LIN {X 0,Y 573.254,Z 377.707,A -85,B 0,C 180,E1 -2096.976,E2 -2096.976} C_VEL
LIN {X 0,Y 573.253,Z 377.7,A -85,B 0,C 180,E1 -2099.488,E2 -2099.488} C_VEL
LIN {X 0,Y 573.258,Z 377.706,A -85,B 0,C 180,E1 -2102.645,E2 -2102.645} C_VEL
LIN {X 0,Y 573.214,Z 377.706,A -85,B 0,C 180,E1 -2105.188,E2 -2105.188} C_VEL
LIN {X 0,Y 573.24,Z 377.699,A -85,B 0,C 180,E1 -2107.808,E2 -2107.808} C_VEL
LIN {X 0,Y 573.25,Z 377.708,A -85,B 0,C 180,E1 -2110.525,E2 -2110.525} C_VEL
LIN {X 0,Y 573.244,Z 377.699,A -85,B 0,C 180,E1 -2113.359,E2 -2113.359} C_VEL
LIN {X 0,Y 573.258,Z 377.706,A -85,B 0,C 180,E1 -2116.33,E2 -2116.33} C_VEL
LIN {X 0,Y 573.264,Z 377.696,A -85,B 0,C 180,E1 -2119.476,E2 -2119.476} C_VEL
LIN {X 0,Y 573.242,Z 377.706,A -85,B 0,C 180,E1 -2122.193,E2 -2122.193} C_VEL
LIN {X 0,Y 573.257,Z 377.698,A -85,B 0,C 180,E1 -2124.815,E2 -2124.815} C_VEL
LIN {X 0,Y 573.258,Z 377.698,A -85,B 0,C 180,E1 -2127.355,E2 -2127.355} C_VEL
LIN {X 0,Y 573.25,Z 377.694,A -85,B 0,C 180,E1 -2130.512,E2 -2130.512} C_VEL
LIN {X 0,Y 573.254,Z 377.697,A -85,B 0,C 180,E1 -2133.024,E2 -2133.024} C_VEL
LIN {X 0,Y 573.277,Z 377.699,A -85,B 0,C 180,E1 -2135.366,E2 -2135.366} C_VEL
LIN {X 0,Y 573.233,Z 377.701,A -85,B 0,C 180,E1 -2138.419,E2 -2138.419} C_VEL
LIN {X 0,Y 573.272,Z 377.696,A -85,B 0,C 180,E1 -2140.731,E2 -2140.731} C_VEL
LIN {X 0,Y 573.253,Z 377.706,A -85,B 0,C 180,E1 -2143.622,E2 -2143.622} C_VEL
LIN {X 0,Y 573.255,Z 377.7,A -85,B 0,C 180,E1 -2146.485,E2 -2146.485} C_VEL
LIN {X 0,Y 574.102,Z 381.406,A -85,B 0,C 180,E1 -2146.64,E2 -2146.64} C_VEL
LIN {X 0,Y 573.92,Z 396.904,A -85,B 0,C 180,E1 -2147.266,E2 -2147.266} C_VEL
LIN {X 0,Y 573.779,Z 408.749,A -85,B 0,C 180,E1 -2147.892,E2 -2147.892} C_VEL
LIN {X 0,Y 573.607,Z 419.401,A -85,B 0,C 180,E1 -2148.575,E2 -2148.575} C_VEL
LIN {X 0,Y 573.485,Z 431.28,A -85,B 0,C 180,E1 -2149.497,E2 -2149.497} C_VEL
LIN {X 0,Y 573.374,Z 441.636,A -85,B 0,C 180,E1 -2150.475,E2 -2150.475} C_VEL
LIN {X 0,Y 573.236,Z 450.947,A -85,B 0,C 180,E1 -2151.54,E2 -2151.54} C_VEL
LIN {X 0,Y 573.142,Z 458.728,A -85,B 0,C 180,E1 -2152.602,E2 -2152.602} C_VEL
LIN {X 0,Y 573.084,Z 465.205,A -85,B 0,C 180,E1 -2153.663,E2 -2153.663} C_VEL
LIN {X 0,Y 573.009,Z 470.597,A -85,B 0,C 180,E1 -2154.722,E2 -2154.722} C_VEL
LIN {X 0,Y 573.038,Z 476.255,A -85,B 0,C 180,E1 -2156.132,E2 -2156.132} C_VEL
LIN {X 0,Y 572.964,Z 479.465,A -85,B 0,C 180,E1 -2157.188,E2 -2157.188} C_VEL
LIN {X 0,Y 572.942,Z 482.451,A -85,B 0,C 180,E1 -2158.594,E2 -2158.594} C_VEL
LIN {X 0,Y 572.936,Z 484.094,A -85,B 0,C 180,E1 -2160,E2 -2160} C_VEL
LIN {X 0,Y 572.945,Z 484.433,A -85,B 0,C 180,E1 -2161.406,E2 -2161.406} C_VEL
LIN {X 0,Y 572.955,Z 483.443,A -85,B 0,C 180,E1 -2162.812,E2 -2162.812} C_VEL
LIN {X 0,Y 573.007,Z 481.089,A -85,B 0,C 180,E1 -2164.22,E2 -2164.22} C_VEL
LIN {X 0,Y 572.994,Z 478.392,A -85,B 0,C 180,E1 -2165.278,E2 -2165.278} C_VEL
LIN {X 0,Y 573.03,Z 473.984,A -85,B 0,C 180,E1 -2166.568,E2 -2166.568} C_VEL
LIN {X 0,Y 573.062,Z 468.762,A -85,B 0,C 180,E1 -2167.753,E2 -2167.753} C_VEL
LIN {X 0,Y 573.131,Z 460.802,A -85,B 0,C 180,E1 -2169.173,E2 -2169.173} C_VEL
LIN {X 0,Y 573.233,Z 451.987,A -85,B 0,C 180,E1 -2170.419,E2 -2170.419} C_VEL
LIN {X 0,Y 573.33,Z 442.788,A -85,B 0,C 180,E1 -2171.49,E2 -2171.49} C_VEL
LIN {X 0,Y 573.474,Z 431.634,A -85,B 0,C 180,E1 -2172.564,E2 -2172.564} C_VEL
LIN {X 0,Y 573.638,Z 420.168,A -85,B 0,C 180,E1 -2173.461,E2 -2173.461} C_VEL
LIN {X 0,Y 573.788,Z 409.059,A -85,B 0,C 180,E1 -2174.18,E2 -2174.18} C_VEL
LIN {X 0,Y 573.948,Z 396.515,A -85,B 0,C 180,E1 -2174.843,E2 -2174.843} C_VEL
LIN {X 0,Y 574.119,Z 381.65,A -85,B 0,C 180,E1 -2175.441,E2 -2175.441} C_VEL
LIN {X 0,Y 573.281,Z 377.703,A -85,B 0,C 180,E1 -2175.601,E2 -2175.601} C_VEL
LIN {X 0,Y 573.24,Z 377.706,A -85,B 0,C 180,E1 -2178.588,E2 -2178.588} C_VEL
LIN {X 0,Y 573.254,Z 377.705,A -85,B 0,C 180,E1 -2181.291,E2 -2181.291} C_VEL
LIN {X 0,Y 573.237,Z 377.708,A -85,B 0,C 180,E1 -2183.865,E2 -2183.865} C_VEL
LIN {X 0,Y 573.239,Z 377.709,A -85,B 0,C 180,E1 -2186.492,E2 -2186.492} C_VEL
LIN {X 0,Y 573.241,Z 377.705,A -85,B 0,C 180,E1 -2188.564,E2 -2188.564} C_VEL
LIN {X 0,Y 573.228,Z 377.707,A -85,B 0,C 180,E1 -2190.993,E2 -2190.993} C_VEL
LIN {X 0,Y 573.265,Z 377.702,A -85,B 0,C 180,E1 -2193.524,E2 -2193.524} C_VEL
LIN {X 0,Y 573.217,Z 377.709,A -85,B 0,C 180,E1 -2196.051,E2 -2196.051} C_VEL
LIN {X 0,Y 573.246,Z 377.706,A -85,B 0,C 180,E1 -2198.701,E2 -2198.701} C_VEL
LIN {X 0,Y 573.256,Z 377.707,A -85,B 0,C 180,E1 -2201.595,E2 -2201.595} C_VEL
LIN {X 0,Y 573.24,Z 377.708,A -85,B 0,C 180,E1 -2204.333,E2 -2204.333} C_VEL
LIN {X 0,Y 573.244,Z 377.707,A -85,B 0,C 180,E1 -2207.358,E2 -2207.358} C_VEL
LIN {X 0,Y 573.25,Z 377.708,A -85,B 0,C 180,E1 -2210.393,E2 -2210.393} C_VEL
LIN {X 0,Y 573.297,Z 377.786,A -85,B 0,C 180,E1 -2211.559,E2 -2211.559} C_VEL
LIN {X 0,Y 573.618,Z 382.639,A -85,B 0,C 180,E1 -2212.544,E2 -2212.544} C_VEL
LIN {X 0,Y 573.399,Z 396.627,A -85,B 0,C 180,E1 -2215.205,E2 -2215.205} C_VEL
LIN {X 0,Y 573.719,Z 413.144,A -85,B 0,C 180,E1 -2218.214,E2 -2218.214} C_VEL
LIN {X 0,Y 573.944,Z 428.097,A -85,B 0,C 180,E1 -2220.873,E2 -2220.873} C_VEL
LIN {X 0,Y 573.98,Z 435.882,A -85,B 0,C 180,E1 -2222.271,E2 -2222.271} C_VEL
LIN {X 0,Y 573.829,Z 449.3,A -85,B 0,C 180,E1 -2225.001,E2 -2225.001} C_VEL
LIN {X 0,Y 573.65,Z 462.702,A -85,B 0,C 180,E1 -2227.679,E2 -2227.679} C_VEL
LIN {X 0,Y 573.5,Z 478.001,A -85,B 0,C 180,E1 -2230.678,E2 -2230.678} C_VEL
LIN {X 0,Y 573.329,Z 493.301,A -85,B 0,C 180,E1 -2233.623,E2 -2233.623} C_VEL
LIN {X 0,Y 573.293,Z 499.756,A -85,B 0,C 180,E1 -2234.854,E2 -2234.854} C_VEL
LIN {X 0,Y 574.29,Z 505.581,A -85,B 0,C 180,E1 -2234.972,E2 -2234.972} C_VEL
LIN {X 0,Y 574.206,Z 520.02,A -85,B 0,C 180,E1 -2235.26,E2 -2235.26} C_VEL
LIN {X 0,Y 574.112,Z 533.209,A -85,B 0,C 180,E1 -2235.66,E2 -2235.66} C_VEL
LIN {X 0,Y 573.972,Z 546.119,A -85,B 0,C 180,E1 -2236.186,E2 -2236.186} C_VEL
LIN {X 0,Y 573.764,Z 558.206,A -85,B 0,C 180,E1 -2236.812,E2 -2236.812} C_VEL
LIN {X 0,Y 573.616,Z 570.7,A -85,B 0,C 180,E1 -2237.618,E2 -2237.618} C_VEL
LIN {X 0,Y 573.481,Z 582.004,A -85,B 0,C 180,E1 -2238.513,E2 -2238.513} C_VEL
LIN {X 0,Y 573.334,Z 593.075,A -85,B 0,C 180,E1 -2239.583,E2 -2239.583} C_VEL
LIN {X 0,Y 573.225,Z 602.195,A -85,B 0,C 180,E1 -2240.65,E2 -2240.65} C_VEL
LIN {X 0,Y 573.128,Z 610.917,A -85,B 0,C 180,E1 -2241.893,E2 -2241.893} C_VEL
LIN {X 0,Y 573.054,Z 617.049,A -85,B 0,C 180,E1 -2242.955,E2 -2242.955} C_VEL
LIN {X 0,Y 573.057,Z 622.132,A -85,B 0,C 180,E1 -2244.016,E2 -2244.016} C_VEL
LIN {X 0,Y 573.024,Z 627.381,A -85,B 0,C 180,E1 -2245.427,E2 -2245.427} C_VEL
LIN {X 0,Y 573.008,Z 630.315,A -85,B 0,C 180,E1 -2246.483,E2 -2246.483} C_VEL
LIN {X 0,Y 572.937,Z 633,A -85,B 0,C 180,E1 -2247.89,E2 -2247.89} C_VEL
LIN {X 0,Y 572.938,Z 634.332,A -85,B 0,C 180,E1 -2249.296,E2 -2249.296} C_VEL
LIN {X 0,Y 572.938,Z 634.333,A -85,B 0,C 180,E1 -2250.702,E2 -2250.702} C_VEL
LIN {X 0,Y 572.937,Z 633.002,A -85,B 0,C 180,E1 -2252.108,E2 -2252.108} C_VEL
LIN {X 0,Y 573.008,Z 630.318,A -85,B 0,C 180,E1 -2253.515,E2 -2253.515} C_VEL
LIN {X 0,Y 572.955,Z 626.203,A -85,B 0,C 180,E1 -2254.925,E2 -2254.925} C_VEL
LIN {X 0,Y 573.049,Z 622.139,A -85,B 0,C 180,E1 -2255.983,E2 -2255.983} C_VEL
LIN {X 0,Y 573.053,Z 617.057,A -85,B 0,C 180,E1 -2257.044,E2 -2257.044} C_VEL
LIN {X 0,Y 573.141,Z 609.805,A -85,B 0,C 180,E1 -2258.283,E2 -2258.283} C_VEL
LIN {X 0,Y 573.252,Z 600.83,A -85,B 0,C 180,E1 -2259.526,E2 -2259.526} C_VEL
LIN {X 0,Y 573.354,Z 591.4,A -85,B 0,C 180,E1 -2260.594,E2 -2260.594} C_VEL
LIN {X 0,Y 573.479,Z 581.068,A -85,B 0,C 180,E1 -2261.566,E2 -2261.566} C_VEL
LIN {X 0,Y 573.635,Z 569.445,A -85,B 0,C 180,E1 -2262.47,E2 -2262.47} C_VEL
LIN {X 0,Y 573.802,Z 556.661,A -85,B 0,C 180,E1 -2263.276,E2 -2263.276} C_VEL
LIN {X 0,Y 573.96,Z 544.18,A -85,B 0,C 180,E1 -2263.903,E2 -2263.903} C_VEL
LIN {X 0,Y 574.135,Z 530.054,A -85,B 0,C 180,E1 -2264.45,E2 -2264.45} C_VEL
LIN {X 0,Y 574.223,Z 516.148,A -85,B 0,C 180,E1 -2264.835,E2 -2264.835} C_VEL
LIN {X 0,Y 574.186,Z 504.665,A -85,B 0,C 180,E1 -2265.045,E2 -2265.045} C_VEL
LIN {X 0,Y 573.291,Z 499.764,A -85,B 0,C 180,E1 -2265.145,E2 -2265.145} C_VEL
LIN {X 0,Y 573.456,Z 483.747,A -85,B 0,C 180,E1 -2268.21,E2 -2268.21} C_VEL
LIN {X 0,Y 573.563,Z 468.92,A -85,B 0,C 180,E1 -2271.096,E2 -2271.096} C_VEL
LIN {X 0,Y 573.734,Z 455.06,A -85,B 0,C 180,E1 -2273.842,E2 -2273.842} C_VEL
LIN {X 0,Y 573.949,Z 441.243,A -85,B 0,C 180,E1 -2276.635,E2 -2276.635} C_VEL
LIN {X 0,Y 574.03,Z 427.742,A -85,B 0,C 180,E1 -2279.322,E2 -2279.322} C_VEL
LIN {X 0,Y 574.031,Z 413.976,A -85,B 0,C 180,E1 -2282.061,E2 -2282.061} C_VEL
LIN {X 0,Y 574.097,Z 400.387,A -85,B 0,C 180,E1 -2284.895,E2 -2284.895} C_VEL
LIN {X 0,Y 574.322,Z 389.132,A -85,B 0,C 180,E1 -2287.306,E2 -2287.306} C_VEL
LIN {X 0,Y 574.322,Z 383.248,A -85,B 0,C 180,E1 -2288.614,E2 -2288.614} C_VEL
LIN {X 0,Y 573.248,Z 377.708,A -85,B 0,C 180,E1 -2289.977,E2 -2289.977} C_VEL
LIN {X 0,Y 573.236,Z 377.701,A -85,B 0,C 180,E1 -2292.641,E2 -2292.641} C_VEL
LIN {X 0,Y 573.232,Z 377.709,A -85,B 0,C 180,E1 -2295.666,E2 -2295.666} C_VEL
LIN {X 0,Y 573.253,Z 377.699,A -85,B 0,C 180,E1 -2298.545,E2 -2298.545} C_VEL
LIN {X 0,Y 573.242,Z 377.703,A -85,B 0,C 180,E1 -2301.298,E2 -2301.298} C_VEL
LIN {X 0,Y 573.256,Z 377.703,A -85,B 0,C 180,E1 -2304.01,E2 -2304.01} C_VEL
LIN {X 0,Y 573.276,Z 377.695,A -85,B 0,C 180,E1 -2306.518,E2 -2306.518} C_VEL
LIN {X 0,Y 573.235,Z 377.702,A -85,B 0,C 180,E1 -2309.114,E2 -2309.114} C_VEL
LIN {X 0,Y 573.255,Z 377.703,A -85,B 0,C 180,E1 -2311.968,E2 -2311.968} C_VEL
LIN {X 0,Y 573.247,Z 377.699,A -85,B 0,C 180,E1 -2314.59,E2 -2314.59} C_VEL
LIN {X 0,Y 573.23,Z 377.709,A -85,B 0,C 180,E1 -2317.662,E2 -2317.662} C_VEL
LIN {X 0,Y 573.248,Z 377.704,A -85,B 0,C 180,E1 -2319.923,E2 -2319.923} C_VEL
LIN {X 0,Y 573.254,Z 377.699,A -85,B 0,C 180,E1 -2322.988,E2 -2322.988} C_VEL
LIN {X 0,Y 573.263,Z 377.703,A -85,B 0,C 180,E1 -2325.807,E2 -2325.807} C_VEL
LIN {X 0,Y 573.272,Z 377.696,A -85,B 0,C 180,E1 -2328.734,E2 -2328.734} C_VEL
LIN {X 0,Y 573.298,Z 377.701,A -85,B 0,C 180,E1 -2331.541,E2 -2331.541} C_VEL
LIN {X 0,Y 573.284,Z 377.694,A -85,B 0,C 180,E1 -2334.372,E2 -2334.372} C_VEL
LIN {X 0,Y 573.3,Z 377.696,A -85,B 0,C 180,E1 -2337.893,E2 -2337.893} C_VEL
LIN {X 0,Y 573.329,Z 377.689,A -85,B 0,C 180,E1 -2340.703,E2 -2340.703} C_VEL
LIN {X 0,Y 573.234,Z 377.709,A -85,B 0,C 180,E1 -2343.515,E2 -2343.515} C_VEL
LIN {X 0,Y 573.285,Z 377.701,A -85,B 0,C 180,E1 -2345.628,E2 -2345.628} C_VEL
LIN {X 0,Y 573.298,Z 377.692,A -85,B 0,C 180,E1 -2348.46,E2 -2348.46} C_VEL
LIN {X 0,Y 573.289,Z 377.703,A -85,B 0,C 180,E1 -2351.312,E2 -2351.312} C_VEL
LIN {X 0,Y 573.271,Z 377.696,A -85,B 0,C 180,E1 -2354.425,E2 -2354.425} C_VEL
LIN {X 0,Y 573.252,Z 377.704,A -85,B 0,C 180,E1 -2357.112,E2 -2357.112} C_VEL
LIN {X 0,Y 573.249,Z 377.699,A -85,B 0,C 180,E1 -2360.077,E2 -2360.077} C_VEL
LIN {X 0,Y 573.231,Z 377.701,A -85,B 0,C 180,E1 -2362.338,E2 -2362.338} C_VEL
LIN {X 0,Y 573.243,Z 377.699,A -85,B 0,C 180,E1 -2364.401,E2 -2364.401} C_VEL
LIN {X 0,Y 572.618,Z 377.784,A -85,B 0,C 180,E1 -2364.988,E2 -2364.988} C_VEL
LIN {X 0,Y 569.781,Z 378.141,A -85,B 0,C 180,E1 -2365.939,E2 -2365.939} C_VEL
LIN {X 0,Y 567.353,Z 378.445,A -85,B 0,C 180,E1 -2366.705,E2 -2366.705} C_VEL
LIN {X 0,Y 566.3,Z 378.573,A -85,B 0,C 180,E1 -2367.296,E2 -2367.296} C_VEL
LIN {X 0,Y 566.211,Z 378.581,A -85,B 0,C 180,E1 -2367.497,E2 -2367.497} C_VEL
LIN {X 0,Y 566.181,Z 378.58,A -85,B 0,C 180,E1 -2370.593,E2 -2370.593} C_VEL
LIN {X 0,Y 566.222,Z 378.582,A -85,B 0,C 180,E1 -2373.102,E2 -2373.102} C_VEL
LIN {X 0,Y 566.205,Z 378.579,A -85,B 0,C 180,E1 -2375.689,E2 -2375.689} C_VEL
LIN {X 0,Y 566.211,Z 378.577,A -85,B 0,C 180,E1 -2378.56,E2 -2378.56} C_VEL
LIN {X 0,Y 566.207,Z 378.585,A -85,B 0,C 180,E1 -2381.137,E2 -2381.137} C_VEL
LIN {X 0,Y 566.196,Z 378.577,A -85,B 0,C 180,E1 -2384.036,E2 -2384.036} C_VEL
LIN {X 0,Y 566.201,Z 378.586,A -85,B 0,C 180,E1 -2387.084,E2 -2387.084} C_VEL
LIN {X 0,Y 566.224,Z 378.575,A -85,B 0,C 180,E1 -2389.804,E2 -2389.804} C_VEL
LIN {X 0,Y 566.197,Z 378.58,A -85,B 0,C 180,E1 -2392.6,E2 -2392.6} C_VEL
LIN {X 0,Y 566.22,Z 378.582,A -85,B 0,C 180,E1 -2395.184,E2 -2395.184} C_VEL
LIN {X 0,Y 566.233,Z 378.574,A -85,B 0,C 180,E1 -2397.745,E2 -2397.745} C_VEL
LIN {X 0,Y 566.204,Z 378.577,A -85,B 0,C 180,E1 -2400.329,E2 -2400.329} C_VEL
LIN {X 0,Y 566.211,Z 378.58,A -85,B 0,C 180,E1 -2402.662,E2 -2402.662} C_VEL
LIN {X 0,Y 566.237,Z 378.58,A -85,B 0,C 180,E1 -2405.04,E2 -2405.04} C_VEL
LIN {X 0,Y 566.195,Z 378.578,A -85,B 0,C 180,E1 -2408.139,E2 -2408.139} C_VEL
LIN {X 0,Y 566.232,Z 378.577,A -85,B 0,C 180,E1 -2410.615,E2 -2410.615} C_VEL
LIN {X 0,Y 566.213,Z 378.578,A -85,B 0,C 180,E1 -2413.413,E2 -2413.413} C_VEL
LIN {X 0,Y 566.148,Z 378.589,A -85,B 0,C 180,E1 -2415.626,E2 -2415.626} C_VEL
LIN {X 0,Y 565.905,Z 378.62,A -85,B 0,C 180,E1 -2417.813,E2 -2417.813} C_VEL
LIN {X 0,Y 565.89,Z 379.999,A -85,B 0,C 180,E1 -2419.265,E2 -2419.265} C_VEL
LIN {X 0,Y 565.884,Z 381.412,A -85,B 0,C 180,E1 -2420.439,E2 -2420.439} C_VEL
LIN {X 0,Y 566.876,Z 389.153,A -85,B 0,C 180,E1 -2420.636,E2 -2420.636} C_VEL
LIN {X 0,Y 566.813,Z 401.962,A -85,B 0,C 180,E1 -2421.04,E2 -2421.04} C_VEL
LIN {X 0,Y 566.692,Z 413.365,A -85,B 0,C 180,E1 -2421.532,E2 -2421.532} C_VEL
LIN {X 0,Y 566.538,Z 424.558,A -85,B 0,C 180,E1 -2422.158,E2 -2422.158} C_VEL
LIN {X 0,Y 566.35,Z 434.772,A -85,B 0,C 180,E1 -2422.872,E2 -2422.872} C_VEL
LIN {X 0,Y 566.194,Z 445.092,A -85,B 0,C 180,E1 -2423.766,E2 -2423.766} C_VEL
LIN {X 0,Y 566.185,Z 453.504,A -85,B 0,C 180,E1 -2424.659,E2 -2424.659} C_VEL
LIN {X 0,Y 566.078,Z 461.71,A -85,B 0,C 180,E1 -2425.729,E2 -2425.729} C_VEL
LIN {X 0,Y 566.012,Z 468.322,A -85,B 0,C 180,E1 -2426.798,E2 -2426.798} C_VEL
LIN {X 0,Y 565.885,Z 473.611,A -85,B 0,C 180,E1 -2427.866,E2 -2427.866} C_VEL
LIN {X 0,Y 565.912,Z 477.737,A -85,B 0,C 180,E1 -2428.933,E2 -2428.933} C_VEL
LIN {X 0,Y 565.843,Z 480.822,A -85,B 0,C 180,E1 -2430.001,E2 -2430.001} C_VEL
LIN {X 0,Y 565.841,Z 482.356,A -85,B 0,C 180,E1 -2430.712,E2 -2430.712} C_VEL
LIN {X 0,Y 565.848,Z 483.465,A -85,B 0,C 180,E1 -2431.424,E2 -2431.424} C_VEL
LIN {X 0,Y 565.873,Z 484.463,A -85,B 0,C 180,E1 -2432.848,E2 -2432.848} C_VEL
LIN {X 0,Y 565.911,Z 484.392,A -85,B 0,C 180,E1 -2433.561,E2 -2433.561} C_VEL
LIN {X 0,Y 565.913,Z 483.897,A -85,B 0,C 180,E1 -2434.274,E2 -2434.274} C_VEL
LIN {X 0,Y 565.923,Z 481.705,A -85,B 0,C 180,E1 -2435.702,E2 -2435.702} C_VEL
LIN {X 0,Y 565.921,Z 479.663,A -85,B 0,C 180,E1 -2436.535,E2 -2436.535} C_VEL
LIN {X 0,Y 565.928,Z 475.173,A -85,B 0,C 180,E1 -2437.852,E2 -2437.852} C_VEL
LIN {X 0,Y 565.966,Z 470.257,A -85,B 0,C 180,E1 -2438.93,E2 -2438.93} C_VEL
LIN {X 0,Y 566.037,Z 464.05,A -85,B 0,C 180,E1 -2440.011,E2 -2440.011} C_VEL
LIN {X 0,Y 566.11,Z 456.152,A -85,B 0,C 180,E1 -2441.11,E2 -2441.11} C_VEL
LIN {X 0,Y 566.224,Z 446.537,A -85,B 0,C 180,E1 -2442.182,E2 -2442.182} C_VEL
LIN {X 0,Y 566.332,Z 437.519,A -85,B 0,C 180,E1 -2442.999,E2 -2442.999} C_VEL
LIN {X 0,Y 566.475,Z 426.339,A -85,B 0,C 180,E1 -2443.818,E2 -2443.818} C_VEL
LIN {X 0,Y 566.652,Z 413.938,A -85,B 0,C 180,E1 -2444.53,E2 -2444.53} C_VEL
LIN {X 0,Y 566.772,Z 401.844,A -85,B 0,C 180,E1 -2445.055,E2 -2445.055} C_VEL
LIN {X 0,Y 566.89,Z 388.921,A -85,B 0,C 180,E1 -2445.459,E2 -2445.459} C_VEL
LIN {X 0,Y 565.865,Z 381.414,A -85,B 0,C 180,E1 -2445.65,E2 -2445.65} C_VEL
LIN {X 0,Y 565.865,Z 378.624,A -85,B 0,C 180,E1 -2448.09,E2 -2448.09} C_VEL
LIN {X 0,Y 566.172,Z 378.589,A -85,B 0,C 180,E1 -2451.1,E2 -2451.1} C_VEL
LIN {X 0,Y 566.173,Z 378.585,A -85,B 0,C 180,E1 -2453.405,E2 -2453.405} C_VEL
LIN {X 0,Y 566.217,Z 378.575,A -85,B 0,C 180,E1 -2455.749,E2 -2455.749} C_VEL
LIN {X 0,Y 566.209,Z 378.576,A -85,B 0,C 180,E1 -2458.202,E2 -2458.202} C_VEL
LIN {X 0,Y 566.196,Z 378.584,A -85,B 0,C 180,E1 -2461.076,E2 -2461.076} C_VEL
LIN {X 0,Y 566.203,Z 378.577,A -85,B 0,C 180,E1 -2463.732,E2 -2463.732} C_VEL
LIN {X 0,Y 566.205,Z 378.585,A -85,B 0,C 180,E1 -2466.57,E2 -2466.57} C_VEL
LIN {X 0,Y 566.221,Z 378.573,A -85,B 0,C 180,E1 -2469.686,E2 -2469.686} C_VEL
LIN {X 0,Y 566.207,Z 378.578,A -85,B 0,C 180,E1 -2472.917,E2 -2472.917} C_VEL
LIN {X 0,Y 566.208,Z 378.58,A -85,B 0,C 180,E1 -2476.048,E2 -2476.048} C_VEL
LIN {X 0,Y 566.217,Z 378.575,A -85,B 0,C 180,E1 -2478.864,E2 -2478.864} C_VEL
LIN {X 0,Y 566.194,Z 378.575,A -85,B 0,C 180,E1 -2481.637,E2 -2481.637} C_VEL
LIN {X 0,Y 566.209,Z 378.581,A -85,B 0,C 180,E1 -2484.311,E2 -2484.311} C_VEL
LIN {X 0,Y 566.224,Z 378.573,A -85,B 0,C 180,E1 -2486.898,E2 -2486.898} C_VEL
LIN {X 0,Y 566.184,Z 378.577,A -85,B 0,C 180,E1 -2489.407,E2 -2489.407} C_VEL
LIN {X 0,Y 566.216,Z 378.579,A -85,B 0,C 180,E1 -2491.857,E2 -2491.857} C_VEL
LIN {X 0,Y 566.216,Z 378.577,A -85,B 0,C 180,E1 -2494.251,E2 -2494.251} C_VEL
LIN {X 0,Y 566.172,Z 378.58,A -85,B 0,C 180,E1 -2496.719,E2 -2496.719} C_VEL
LIN {X 0,Y 566.211,Z 378.584,A -85,B 0,C 180,E1 -2499.662,E2 -2499.662} C_VEL
LIN {X 0,Y 566.203,Z 378.577,A -85,B 0,C 180,E1 -2502.668,E2 -2502.668} C_VEL
LIN {X 0,Y 566.237,Z 378.58,A -85,B 0,C 180,E1 -2505.627,E2 -2505.627} C_VEL
LIN {X 0,Y 566.243,Z 378.574,A -85,B 0,C 180,E1 -2506.337,E2 -2506.337} C_VEL
LIN {X 0,Y 567.199,Z 383.09,A -85,B 0,C 180,E1 -2506.52,E2 -2506.52} C_VEL
LIN {X 0,Y 567.013,Z 397.155,A -85,B 0,C 180,E1 -2507.108,E2 -2507.108} C_VEL
LIN {X 0,Y 566.831,Z 408.959,A -85,B 0,C 180,E1 -2507.741,E2 -2507.741} C_VEL
LIN {X 0,Y 566.643,Z 420.143,A -85,B 0,C 180,E1 -2508.472,E2 -2508.472} C_VEL
LIN {X 0,Y 566.474,Z 432.48,A -85,B 0,C 180,E1 -2509.455,E2 -2509.455} C_VEL
LIN {X 0,Y 566.302,Z 443.378,A -85,B 0,C 180,E1 -2510.535,E2 -2510.535} C_VEL
LIN {X 0,Y 566.165,Z 452.441,A -85,B 0,C 180,E1 -2511.613,E2 -2511.613} C_VEL
LIN {X 0,Y 566.05,Z 461.134,A -85,B 0,C 180,E1 -2512.868,E2 -2512.868} C_VEL
LIN {X 0,Y 566.003,Z 468.971,A -85,B 0,C 180,E1 -2514.299,E2 -2514.299} C_VEL
LIN {X 0,Y 565.964,Z 473.658,A -85,B 0,C 180,E1 -2515.37,E2 -2515.37} C_VEL
LIN {X 0,Y 565.933,Z 477.425,A -85,B 0,C 180,E1 -2516.44,E2 -2516.44} C_VEL
LIN {X 0,Y 565.883,Z 479.499,A -85,B 0,C 180,E1 -2517.152,E2 -2517.152} C_VEL
LIN {X 0,Y 565.842,Z 482.469,A -85,B 0,C 180,E1 -2518.576,E2 -2518.576} C_VEL
LIN {X 0,Y 565.837,Z 483.482,A -85,B 0,C 180,E1 -2519.288,E2 -2519.288} C_VEL
LIN {X 0,Y 565.836,Z 484.441,A -85,B 0,C 180,E1 -2520.711,E2 -2520.711} C_VEL
LIN {X 0,Y 565.835,Z 484.065,A -85,B 0,C 180,E1 -2522.135,E2 -2522.135} C_VEL
LIN {X 0,Y 565.873,Z 483.432,A -85,B 0,C 180,E1 -2522.847,E2 -2522.847} C_VEL
LIN {X 0,Y 565.912,Z 481.052,A -85,B 0,C 180,E1 -2524.273,E2 -2524.273} C_VEL
LIN {X 0,Y 565.92,Z 478.351,A -85,B 0,C 180,E1 -2525.344,E2 -2525.344} C_VEL
LIN {X 0,Y 565.946,Z 474.277,A -85,B 0,C 180,E1 -2526.56,E2 -2526.56} C_VEL
LIN {X 0,Y 565.974,Z 470.388,A -85,B 0,C 180,E1 -2527.492,E2 -2527.492} C_VEL
LIN {X 0,Y 566.022,Z 463.906,A -85,B 0,C 180,E1 -2528.749,E2 -2528.749} C_VEL
LIN {X 0,Y 566.098,Z 457.153,A -85,B 0,C 180,E1 -2529.829,E2 -2529.829} C_VEL
LIN {X 0,Y 566.177,Z 448.723,A -85,B 0,C 180,E1 -2530.949,E2 -2530.949} C_VEL
LIN {X 0,Y 566.346,Z 439.215,A -85,B 0,C 180,E1 -2531.997,E2 -2531.997} C_VEL
LIN {X 0,Y 566.495,Z 429.325,A -85,B 0,C 180,E1 -2532.903,E2 -2532.903} C_VEL
LIN {X 0,Y 566.703,Z 418.675,A -85,B 0,C 180,E1 -2533.72,E2 -2533.72} C_VEL
LIN {X 0,Y 566.864,Z 407.54,A -85,B 0,C 180,E1 -2534.433,E2 -2534.433} C_VEL
LIN {X 0,Y 567.105,Z 394.98,A -85,B 0,C 180,E1 -2535.085,E2 -2535.085} C_VEL
LIN {X 0,Y 567.228,Z 382.575,A -85,B 0,C 180,E1 -2535.587,E2 -2535.587} C_VEL
LIN {X 0,Y 566.214,Z 378.582,A -85,B 0,C 180,E1 -2535.755,E2 -2535.755} C_VEL
LIN {X 0,Y 566.211,Z 378.583,A -85,B 0,C 180,E1 -2538.078,E2 -2538.078} C_VEL
LIN {X 0,Y 566.216,Z 378.585,A -85,B 0,C 180,E1 -2540.337,E2 -2540.337} C_VEL
LIN {X 0,Y 566.193,Z 378.584,A -85,B 0,C 180,E1 -2543.404,E2 -2543.404} C_VEL
LIN {X 0,Y 566.215,Z 378.581,A -85,B 0,C 180,E1 -2545.749,E2 -2545.749} C_VEL
LIN {X 0,Y 566.205,Z 378.582,A -85,B 0,C 180,E1 -2548.202,E2 -2548.202} C_VEL
LIN {X 0,Y 566.193,Z 378.583,A -85,B 0,C 180,E1 -2551.076,E2 -2551.076} C_VEL
LIN {X 0,Y 566.214,Z 378.581,A -85,B 0,C 180,E1 -2553.734,E2 -2553.734} C_VEL
LIN {X 0,Y 566.202,Z 378.585,A -85,B 0,C 180,E1 -2556.57,E2 -2556.57} C_VEL
LIN {X 0,Y 566.218,Z 378.58,A -85,B 0,C 180,E1 -2559.686,E2 -2559.686} C_VEL
LIN {X 0,Y 566.218,Z 378.581,A -85,B 0,C 180,E1 -2562.087,E2 -2562.087} C_VEL
LIN {X 0,Y 566.172,Z 378.588,A -85,B 0,C 180,E1 -2565.036,E2 -2565.036} C_VEL
LIN {X 0,Y 566.214,Z 378.585,A -85,B 0,C 180,E1 -2567.912,E2 -2567.912} C_VEL
LIN {X 0,Y 566.227,Z 378.582,A -85,B 0,C 180,E1 -2570.727,E2 -2570.727} C_VEL
LIN {X 0,Y 566.231,Z 378.656,A -85,B 0,C 180,E1 -2571.403,E2 -2571.403} C_VEL
LIN {X 0,Y 566.639,Z 383.157,A -85,B 0,C 180,E1 -2572.349,E2 -2572.349} C_VEL
LIN {X 0,Y 566.418,Z 396.614,A -85,B 0,C 180,E1 -2574.976,E2 -2574.976} C_VEL
LIN {X 0,Y 566.669,Z 413.918,A -85,B 0,C 180,E1 -2578.19,E2 -2578.19} C_VEL
LIN {X 0,Y 566.889,Z 428.862,A -85,B 0,C 180,E1 -2580.882,E2 -2580.882} C_VEL
LIN {X 0,Y 566.958,Z 444.499,A -85,B 0,C 180,E1 -2583.694,E2 -2583.694} C_VEL
LIN {X 0,Y 566.762,Z 458.877,A -85,B 0,C 180,E1 -2586.621,E2 -2586.621} C_VEL
LIN {X 0,Y 566.53,Z 474.177,A -85,B 0,C 180,E1 -2589.674,E2 -2589.674} C_VEL
LIN {X 0,Y 566.399,Z 487.564,A -85,B 0,C 180,E1 -2592.301,E2 -2592.301} C_VEL
LIN {X 0,Y 566.263,Z 499.756,A -85,B 0,C 180,E1 -2594.661,E2 -2594.661} C_VEL
LIN {X 0,Y 567.443,Z 507.087,A -85,B 0,C 180,E1 -2594.809,E2 -2594.809} C_VEL
LIN {X 0,Y 567.328,Z 521.177,A -85,B 0,C 180,E1 -2595.107,E2 -2595.107} C_VEL
LIN {X 0,Y 567.211,Z 535.029,A -85,B 0,C 180,E1 -2595.546,E2 -2595.546} C_VEL
LIN {X 0,Y 567.049,Z 548.082,A -85,B 0,C 180,E1 -2596.105,E2 -2596.105} C_VEL
LIN {X 0,Y 566.778,Z 561.248,A -85,B 0,C 180,E1 -2596.829,E2 -2596.829} C_VEL
LIN {X 0,Y 566.64,Z 573.134,A -85,B 0,C 180,E1 -2597.645,E2 -2597.645} C_VEL
LIN {X 0,Y 566.445,Z 584.215,A -85,B 0,C 180,E1 -2598.571,E2 -2598.571} C_VEL
LIN {X 0,Y 566.295,Z 594.701,A -85,B 0,C 180,E1 -2599.632,E2 -2599.632} C_VEL
LIN {X 0,Y 566.178,Z 603.554,A -85,B 0,C 180,E1 -2600.713,E2 -2600.713} C_VEL
LIN {X 0,Y 566.047,Z 612.033,A -85,B 0,C 180,E1 -2601.97,E2 -2601.97} C_VEL
LIN {X 0,Y 565.992,Z 619.041,A -85,B 0,C 180,E1 -2603.261,E2 -2603.261} C_VEL
LIN {X 0,Y 565.929,Z 624.958,A -85,B 0,C 180,E1 -2604.655,E2 -2604.655} C_VEL
LIN {X 0,Y 565.956,Z 628.442,A -85,B 0,C 180,E1 -2605.726,E2 -2605.726} C_VEL
LIN {X 0,Y 565.875,Z 631.832,A -85,B 0,C 180,E1 -2607.152,E2 -2607.152} C_VEL
LIN {X 0,Y 565.84,Z 633.832,A -85,B 0,C 180,E1 -2608.576,E2 -2608.576} C_VEL
LIN {X 0,Y 565.837,Z 634.5,A -85,B 0,C 180,E1 -2609.999,E2 -2609.999} C_VEL
LIN {X 0,Y 565.84,Z 633.833,A -85,B 0,C 180,E1 -2611.423,E2 -2611.423} C_VEL
LIN {X 0,Y 565.874,Z 631.833,A -85,B 0,C 180,E1 -2612.847,E2 -2612.847} C_VEL
LIN {X 0,Y 565.956,Z 628.445,A -85,B 0,C 180,E1 -2614.272,E2 -2614.272} C_VEL
LIN {X 0,Y 565.984,Z 623.572,A -85,B 0,C 180,E1 -2615.7,E2 -2615.7} C_VEL
LIN {X 0,Y 565.994,Z 619.049,A -85,B 0,C 180,E1 -2616.738,E2 -2616.738} C_VEL
LIN {X 0,Y 566.046,Z 612.042,A -85,B 0,C 180,E1 -2618.028,E2 -2618.028} C_VEL
LIN {X 0,Y 566.18,Z 603.565,A -85,B 0,C 180,E1 -2619.285,E2 -2619.285} C_VEL
LIN {X 0,Y 566.294,Z 594.715,A -85,B 0,C 180,E1 -2620.366,E2 -2620.366} C_VEL
LIN {X 0,Y 566.483,Z 584.001,A -85,B 0,C 180,E1 -2621.448,E2 -2621.448} C_VEL
LIN {X 0,Y 566.638,Z 573.154,A -85,B 0,C 180,E1 -2622.353,E2 -2622.353} C_VEL
LIN {X 0,Y 566.776,Z 561.271,A -85,B 0,C 180,E1 -2623.17,E2 -2623.17} C_VEL
LIN {X 0,Y 567.051,Z 548.116,A -85,B 0,C 180,E1 -2623.893,E2 -2623.893} C_VEL
LIN {X 0,Y 567.234,Z 535.087,A -85,B 0,C 180,E1 -2624.451,E2 -2624.451} C_VEL
LIN {X 0,Y 567.32,Z 521.304,A -85,B 0,C 180,E1 -2624.89,E2 -2624.89} C_VEL
LIN {X 0,Y 567.44,Z 507.195,A -85,B 0,C 180,E1 -2625.19,E2 -2625.19} C_VEL
LIN {X 0,Y 566.261,Z 499.764,A -85,B 0,C 180,E1 -2625.337,E2 -2625.337} C_VEL
LIN {X 0,Y 566.454,Z 483.747,A -85,B 0,C 180,E1 -2628.443,E2 -2628.443} C_VEL
LIN {X 0,Y 566.597,Z 469.257,A -85,B 0,C 180,E1 -2631.301,E2 -2631.301} C_VEL
LIN {X 0,Y 566.76,Z 456.974,A -85,B 0,C 180,E1 -2633.765,E2 -2633.765} C_VEL
LIN {X 0,Y 566.98,Z 443.497,A -85,B 0,C 180,E1 -2636.501,E2 -2636.501} C_VEL
LIN {X 0,Y 567.06,Z 428.236,A -85,B 0,C 180,E1 -2639.514,E2 -2639.514} C_VEL
LIN {X 0,Y 567.139,Z 413.075,A -85,B 0,C 180,E1 -2642.578,E2 -2642.578} C_VEL
LIN {X 0,Y 567.305,Z 397.083,A -85,B 0,C 180,E1 -2645.988,E2 -2645.988} C_VEL
LIN {X 0,Y 567.532,Z 386.835,A -85,B 0,C 180,E1 -2648.254,E2 -2648.254} C_VEL
LIN {X 0,Y 566.872,Z 381.704,A -85,B 0,C 180,E1 -2649.468,E2 -2649.468} C_VEL
LIN {X 0,Y 566.22,Z 378.583,A -85,B 0,C 180,E1 -2650.251,E2 -2650.251} C_VEL
LIN {X 0,Y 566.198,Z 378.579,A -85,B 0,C 180,E1 -2653.053,E2 -2653.053} C_VEL
LIN {X 0,Y 566.196,Z 378.583,A -85,B 0,C 180,E1 -2656.047,E2 -2656.047} C_VEL
LIN {X 0,Y 566.213,Z 378.575,A -85,B 0,C 180,E1 -2658.864,E2 -2658.864} C_VEL
LIN {X 0,Y 566.183,Z 378.587,A -85,B 0,C 180,E1 -2661.637,E2 -2661.637} C_VEL
LIN {X 0,Y 566.203,Z 378.578,A -85,B 0,C 180,E1 -2664.311,E2 -2664.311} C_VEL
LIN {X 0,Y 566.22,Z 378.575,A -85,B 0,C 180,E1 -2666.898,E2 -2666.898} C_VEL
LIN {X 0,Y 566.185,Z 378.584,A -85,B 0,C 180,E1 -2669.408,E2 -2669.408} C_VEL
LIN {X 0,Y 566.218,Z 378.581,A -85,B 0,C 180,E1 -2671.858,E2 -2671.858} C_VEL
LIN {X 0,Y 566.216,Z 378.576,A -85,B 0,C 180,E1 -2674.251,E2 -2674.251} C_VEL
LIN {X 0,Y 566.182,Z 378.579,A -85,B 0,C 180,E1 -2676.713,E2 -2676.713} C_VEL
LIN {X 0,Y 566.211,Z 378.584,A -85,B 0,C 180,E1 -2679.663,E2 -2679.663} C_VEL
LIN {X 0,Y 566.195,Z 378.577,A -85,B 0,C 180,E1 -2682.668,E2 -2682.668} C_VEL
LIN {X 0,Y 566.223,Z 378.582,A -85,B 0,C 180,E1 -2685.627,E2 -2685.627} C_VEL
LIN {X 0,Y 566.264,Z 378.569,A -85,B 0,C 180,E1 -2688.654,E2 -2688.654} C_VEL
LIN {X 0,Y 566.239,Z 378.581,A -85,B 0,C 180,E1 -2691.435,E2 -2691.435} C_VEL
LIN {X 0,Y 566.252,Z 378.571,A -85,B 0,C 180,E1 -2694.302,E2 -2694.302} C_VEL
LIN {X 0,Y 566.272,Z 378.572,A -85,B 0,C 180,E1 -2697.866,E2 -2697.866} C_VEL
LIN {X 0,Y 566.298,Z 378.565,A -85,B 0,C 180,E1 -2700.711,E2 -2700.711} C_VEL
LIN {X 0,Y 566.27,Z 378.57,A -85,B 0,C 180,E1 -2702.846,E2 -2702.846} C_VEL
LIN {X 0,Y 566.253,Z 378.576,A -85,B 0,C 180,E1 -2705.699,E2 -2705.699} C_VEL
LIN {X 0,Y 566.239,Z 378.572,A -85,B 0,C 180,E1 -2708.566,E2 -2708.566} C_VEL
LIN {X 0,Y 566.241,Z 378.58,A -85,B 0,C 180,E1 -2711.455,E2 -2711.455} C_VEL
LIN {X 0,Y 566.224,Z 378.574,A -85,B 0,C 180,E1 -2714.508,E2 -2714.508} C_VEL
LIN {X 0,Y 566.197,Z 378.586,A -85,B 0,C 180,E1 -2717.332,E2 -2717.332} C_VEL
LIN {X 0,Y 566.211,Z 378.575,A -85,B 0,C 180,E1 -2720.338,E2 -2720.338} C_VEL
LIN {X 0,Y 566.181,Z 378.587,A -85,B 0,C 180,E1 -2723.405,E2 -2723.405} C_VEL
LIN {X 0,Y 566.217,Z 378.578,A -85,B 0,C 180,E1 -2725.749,E2 -2725.749} C_VEL
LIN {X 0,Y 566.211,Z 378.581,A -85,B 0,C 180,E1 -2727.497,E2 -2727.497} C_VEL
LIN {X 0,Y 565.53,Z 378.663,A -85,B 0,C 180,E1 -2728.09,E2 -2728.09} C_VEL
LIN {X 0,Y 562.658,Z 379.025,A -85,B 0,C 180,E1 -2729.054,E2 -2729.054} C_VEL
LIN {X 0,Y 560.244,Z 379.321,A -85,B 0,C 180,E1 -2729.829,E2 -2729.829} C_VEL
LIN {X 0,Y 559.217,Z 379.447,A -85,B 0,C 180,E1 -2730.428,E2 -2730.428} C_VEL
LIN {X 0,Y 559.139,Z 379.458,A -85,B 0,C 180,E1 -2730.631,E2 -2730.631} C_VEL
LIN {X 0,Y 559.171,Z 379.457,A -85,B 0,C 180,E1 -2733.575,E2 -2733.575} C_VEL
LIN {X 0,Y 559.163,Z 379.454,A -85,B 0,C 180,E1 -2736.45,E2 -2736.45} C_VEL
LIN {X 0,Y 559.173,Z 379.458,A -85,B 0,C 180,E1 -2738.935,E2 -2738.935} C_VEL
LIN {X 0,Y 559.188,Z 379.452,A -85,B 0,C 180,E1 -2741.768,E2 -2741.768} C_VEL
LIN {X 0,Y 559.136,Z 379.461,A -85,B 0,C 180,E1 -2744.74,E2 -2744.74} C_VEL
LIN {X 0,Y 559.173,Z 379.453,A -85,B 0,C 180,E1 -2747.864,E2 -2747.864} C_VEL
LIN {X 0,Y 559.183,Z 379.451,A -85,B 0,C 180,E1 -2750.136,E2 -2750.136} C_VEL
LIN {X 0,Y 559.145,Z 379.463,A -85,B 0,C 180,E1 -2752.893,E2 -2752.893} C_VEL
LIN {X 0,Y 559.156,Z 379.457,A -85,B 0,C 180,E1 -2755.557,E2 -2755.557} C_VEL
LIN {X 0,Y 559.169,Z 379.453,A -85,B 0,C 180,E1 -2758.139,E2 -2758.139} C_VEL
LIN {X 0,Y 559.143,Z 379.46,A -85,B 0,C 180,E1 -2760.648,E2 -2760.648} C_VEL
LIN {X 0,Y 559.171,Z 379.46,A -85,B 0,C 180,E1 -2763.174,E2 -2763.174} C_VEL
LIN {X 0,Y 559.158,Z 379.457,A -85,B 0,C 180,E1 -2765.496,E2 -2765.496} C_VEL
LIN {X 0,Y 559.173,Z 379.457,A -85,B 0,C 180,E1 -2768.625,E2 -2768.625} C_VEL
LIN {X 0,Y 559.164,Z 379.462,A -85,B 0,C 180,E1 -2770.927,E2 -2770.927} C_VEL
LIN {X 0,Y 559.158,Z 379.454,A -85,B 0,C 180,E1 -2773.949,E2 -2773.949} C_VEL
LIN {X 0,Y 559.042,Z 379.478,A -85,B 0,C 180,E1 -2776.182,E2 -2776.182} C_VEL
LIN {X 0,Y 558.805,Z 379.676,A -85,B 0,C 180,E1 -2778.813,E2 -2778.813} C_VEL
LIN {X 0,Y 558.816,Z 381.405,A -85,B 0,C 180,E1 -2780.271,E2 -2780.271} C_VEL
LIN {X 0,Y 559.933,Z 389.751,A -85,B 0,C 180,E1 -2780.496,E2 -2780.496} C_VEL
LIN {X 0,Y 559.871,Z 402.991,A -85,B 0,C 180,E1 -2780.928,E2 -2780.928} C_VEL
LIN {X 0,Y 559.701,Z 414.146,A -85,B 0,C 180,E1 -2781.425,E2 -2781.425} C_VEL
LIN {X 0,Y 559.548,Z 425.164,A -85,B 0,C 180,E1 -2782.059,E2 -2782.059} C_VEL
LIN {X 0,Y 559.323,Z 435.259,A -85,B 0,C 180,E1 -2782.782,E2 -2782.782} C_VEL
LIN {X 0,Y 559.158,Z 445.496,A -85,B 0,C 180,E1 -2783.687,E2 -2783.687} C_VEL
LIN {X 0,Y 559.141,Z 453.829,A -85,B 0,C 180,E1 -2784.592,E2 -2784.592} C_VEL
LIN {X 0,Y 559.015,Z 461.971,A -85,B 0,C 180,E1 -2785.675,E2 -2785.675} C_VEL
LIN {X 0,Y 558.927,Z 468.532,A -85,B 0,C 180,E1 -2786.757,E2 -2786.757} C_VEL
LIN {X 0,Y 558.792,Z 473.78,A -85,B 0,C 180,E1 -2787.838,E2 -2787.838} C_VEL
LIN {X 0,Y 558.818,Z 477.867,A -85,B 0,C 180,E1 -2788.92,E2 -2788.92} C_VEL
LIN {X 0,Y 558.745,Z 480.916,A -85,B 0,C 180,E1 -2790.001,E2 -2790.001} C_VEL
LIN {X 0,Y 558.742,Z 482.432,A -85,B 0,C 180,E1 -2790.721,E2 -2790.721} C_VEL
LIN {X 0,Y 558.747,Z 483.507,A -85,B 0,C 180,E1 -2791.442,E2 -2791.442} C_VEL
LIN {X 0,Y 558.795,Z 484.471,A -85,B 0,C 180,E1 -2792.884,E2 -2792.884} C_VEL
LIN {X 0,Y 558.82,Z 484.38,A -85,B 0,C 180,E1 -2793.606,E2 -2793.606} C_VEL
LIN {X 0,Y 558.805,Z 483.855,A -85,B 0,C 180,E1 -2794.328,E2 -2794.328} C_VEL
LIN {X 0,Y 558.832,Z 481.628,A -85,B 0,C 180,E1 -2795.775,E2 -2795.775} C_VEL
LIN {X 0,Y 558.82,Z 478.945,A -85,B 0,C 180,E1 -2796.826,E2 -2796.826} C_VEL
LIN {X 0,Y 558.857,Z 475.021,A -85,B 0,C 180,E1 -2797.952,E2 -2797.952} C_VEL
LIN {X 0,Y 558.877,Z 470.062,A -85,B 0,C 180,E1 -2799.045,E2 -2799.045} C_VEL
LIN {X 0,Y 558.98,Z 463.807,A -85,B 0,C 180,E1 -2800.139,E2 -2800.139} C_VEL
LIN {X 0,Y 559.042,Z 455.378,A -85,B 0,C 180,E1 -2801.309,E2 -2801.309} C_VEL
LIN {X 0,Y 559.193,Z 446.151,A -85,B 0,C 180,E1 -2802.337,E2 -2802.337} C_VEL
LIN {X 0,Y 559.386,Z 435.884,A -85,B 0,C 180,E1 -2803.256,E2 -2803.256} C_VEL
LIN {X 0,Y 559.484,Z 425.737,A -85,B 0,C 180,E1 -2803.994,E2 -2803.994} C_VEL
LIN {X 0,Y 559.69,Z 414.467,A -85,B 0,C 180,E1 -2804.648,E2 -2804.648} C_VEL
LIN {X 0,Y 559.839,Z 401.861,A -85,B 0,C 180,E1 -2805.205,E2 -2805.205} C_VEL
LIN {X 0,Y 559.961,Z 389.181,A -85,B 0,C 180,E1 -2805.609,E2 -2805.609} C_VEL
LIN {X 0,Y 558.754,Z 381.393,A -85,B 0,C 180,E1 -2805.831,E2 -2805.831} C_VEL
LIN {X 0,Y 558.758,Z 379.51,A -85,B 0,C 180,E1 -2807.571,E2 -2807.571} C_VEL
LIN {X 0,Y 558.962,Z 379.488,A -85,B 0,C 180,E1 -2809.846,E2 -2809.846} C_VEL
LIN {X 0,Y 559.143,Z 379.456,A -85,B 0,C 180,E1 -2812.153,E2 -2812.153} C_VEL
LIN {X 0,Y 559.182,Z 379.456,A -85,B 0,C 180,E1 -2815.298,E2 -2815.298} C_VEL
LIN {X 0,Y 559.154,Z 379.455,A -85,B 0,C 180,E1 -2817.714,E2 -2817.714} C_VEL
LIN {X 0,Y 559.159,Z 379.455,A -85,B 0,C 180,E1 -2820.183,E2 -2820.183} C_VEL
LIN {X 0,Y 559.158,Z 379.463,A -85,B 0,C 180,E1 -2822.716,E2 -2822.716} C_VEL
LIN {X 0,Y 559.134,Z 379.459,A -85,B 0,C 180,E1 -2825.324,E2 -2825.324} C_VEL
LIN {X 0,Y 559.139,Z 379.457,A -85,B 0,C 180,E1 -2828.018,E2 -2828.018} C_VEL
LIN {X 0,Y 559.161,Z 379.458,A -85,B 0,C 180,E1 -2830.812,E2 -2830.812} C_VEL
LIN {X 0,Y 559.147,Z 379.456,A -85,B 0,C 180,E1 -2833.734,E2 -2833.734} C_VEL
LIN {X 0,Y 559.173,Z 379.455,A -85,B 0,C 180,E1 -2836.801,E2 -2836.801} C_VEL
LIN {X 0,Y 559.182,Z 379.45,A -85,B 0,C 180,E1 -2839.189,E2 -2839.189} C_VEL
LIN {X 0,Y 559.14,Z 379.457,A -85,B 0,C 180,E1 -2841.983,E2 -2841.983} C_VEL
LIN {X 0,Y 559.152,Z 379.455,A -85,B 0,C 180,E1 -2844.785,E2 -2844.785} C_VEL
LIN {X 0,Y 559.16,Z 379.454,A -85,B 0,C 180,E1 -2847.364,E2 -2847.364} C_VEL
LIN {X 0,Y 559.152,Z 379.453,A -85,B 0,C 180,E1 -2850.143,E2 -2850.143} C_VEL
LIN {X 0,Y 559.173,Z 379.45,A -85,B 0,C 180,E1 -2853.098,E2 -2853.098} C_VEL
LIN {X 0,Y 559.159,Z 379.46,A -85,B 0,C 180,E1 -2855.495,E2 -2855.495} C_VEL
LIN {X 0,Y 559.176,Z 379.452,A -85,B 0,C 180,E1 -2858.624,E2 -2858.624} C_VEL
LIN {X 0,Y 559.165,Z 379.455,A -85,B 0,C 180,E1 -2860.926,E2 -2860.926} C_VEL
LIN {X 0,Y 559.169,Z 379.456,A -85,B 0,C 180,E1 -2863.948,E2 -2863.948} C_VEL
LIN {X 0,Y 559.234,Z 379.448,A -85,B 0,C 180,E1 -2866.185,E2 -2866.185} C_VEL
LIN {X 0,Y 560.265,Z 383.482,A -85,B 0,C 180,E1 -2866.35,E2 -2866.35} C_VEL
LIN {X 0,Y 560.109,Z 397.406,A -85,B 0,C 180,E1 -2866.947,E2 -2866.947} C_VEL
LIN {X 0,Y 559.906,Z 409.169,A -85,B 0,C 180,E1 -2867.587,E2 -2867.587} C_VEL
LIN {X 0,Y 559.7,Z 418.912,A -85,B 0,C 180,E1 -2868.226,E2 -2868.226} C_VEL
LIN {X 0,Y 559.58,Z 428.656,A -85,B 0,C 180,E1 -2868.983,E2 -2868.983} C_VEL
LIN {X 0,Y 559.343,Z 438.331,A -85,B 0,C 180,E1 -2869.868,E2 -2869.868} C_VEL
LIN {X 0,Y 559.201,Z 448.282,A -85,B 0,C 180,E1 -2870.961,E2 -2870.961} C_VEL
LIN {X 0,Y 559.065,Z 456.489,A -85,B 0,C 180,E1 -2872.051,E2 -2872.051} C_VEL
LIN {X 0,Y 558.95,Z 463.323,A -85,B 0,C 180,E1 -2873.14,E2 -2873.14} C_VEL
LIN {X 0,Y 558.938,Z 469.026,A -85,B 0,C 180,E1 -2874.227,E2 -2874.227} C_VEL
LIN {X 0,Y 558.87,Z 473.702,A -85,B 0,C 180,E1 -2875.311,E2 -2875.311} C_VEL
LIN {X 0,Y 558.844,Z 477.46,A -85,B 0,C 180,E1 -2876.395,E2 -2876.395} C_VEL
LIN {X 0,Y 558.806,Z 479.533,A -85,B 0,C 180,E1 -2877.116,E2 -2877.116} C_VEL
LIN {X 0,Y 558.742,Z 482.487,A -85,B 0,C 180,E1 -2878.558,E2 -2878.558} C_VEL
LIN {X 0,Y 558.737,Z 483.499,A -85,B 0,C 180,E1 -2879.279,E2 -2879.279} C_VEL
LIN {X 0,Y 558.736,Z 484.445,A -85,B 0,C 180,E1 -2880.721,E2 -2880.721} C_VEL
LIN {X 0,Y 558.742,Z 484.049,A -85,B 0,C 180,E1 -2882.162,E2 -2882.162} C_VEL
LIN {X 0,Y 558.794,Z 483.42,A -85,B 0,C 180,E1 -2882.884,E2 -2882.884} C_VEL
LIN {X 0,Y 558.806,Z 481.015,A -85,B 0,C 180,E1 -2884.328,E2 -2884.328} C_VEL
LIN {X 0,Y 558.845,Z 478.31,A -85,B 0,C 180,E1 -2885.412,E2 -2885.412} C_VEL
LIN {X 0,Y 558.845,Z 474.631,A -85,B 0,C 180,E1 -2886.535,E2 -2886.535} C_VEL
LIN {X 0,Y 558.9,Z 470.318,A -85,B 0,C 180,E1 -2887.587,E2 -2887.587} C_VEL
LIN {X 0,Y 558.962,Z 464.843,A -85,B 0,C 180,E1 -2888.678,E2 -2888.678} C_VEL
LIN {X 0,Y 559.024,Z 458.258,A -85,B 0,C 180,E1 -2889.771,E2 -2889.771} C_VEL
LIN {X 0,Y 559.128,Z 450.353,A -85,B 0,C 180,E1 -2890.868,E2 -2890.868} C_VEL
LIN {X 0,Y 559.297,Z 440.868,A -85,B 0,C 180,E1 -2891.966,E2 -2891.966} C_VEL
LIN {X 0,Y 559.488,Z 430.255,A -85,B 0,C 180,E1 -2892.975,E2 -2892.975} C_VEL
LIN {X 0,Y 559.707,Z 419.767,A -85,B 0,C 180,E1 -2893.802,E2 -2893.802} C_VEL
LIN {X 0,Y 559.885,Z 410.106,A -85,B 0,C 180,E1 -2894.447,E2 -2894.447} C_VEL
LIN {X 0,Y 560.078,Z 400.173,A -85,B 0,C 180,E1 -2895.004,E2 -2895.004} C_VEL
LIN {X 0,Y 560.233,Z 389.253,A -85,B 0,C 180,E1 -2895.507,E2 -2895.507} C_VEL
LIN {X 0,Y 560.266,Z 383.495,A -85,B 0,C 180,E1 -2895.739,E2 -2895.739} C_VEL
LIN {X 0,Y 559.183,Z 379.458,A -85,B 0,C 180,E1 -2895.911,E2 -2895.911} C_VEL
LIN {X 0,Y 559.157,Z 379.461,A -85,B 0,C 180,E1 -2898.314,E2 -2898.314} C_VEL
LIN {X 0,Y 559.182,Z 379.459,A -85,B 0,C 180,E1 -2900.604,E2 -2900.604} C_VEL
LIN {X 0,Y 559.15,Z 379.462,A -85,B 0,C 180,E1 -2903.716,E2 -2903.716} C_VEL
LIN {X 0,Y 559.183,Z 379.457,A -85,B 0,C 180,E1 -2906.097,E2 -2906.097} C_VEL
LIN {X 0,Y 559.166,Z 379.458,A -85,B 0,C 180,E1 -2908.529,E2 -2908.529} C_VEL
LIN {X 0,Y 559.149,Z 379.462,A -85,B 0,C 180,E1 -2911.273,E2 -2911.273} C_VEL
LIN {X 0,Y 559.168,Z 379.461,A -85,B 0,C 180,E1 -2913.949,E2 -2913.949} C_VEL
LIN {X 0,Y 559.144,Z 379.462,A -85,B 0,C 180,E1 -2917.108,E2 -2917.108} C_VEL
LIN {X 0,Y 559.164,Z 379.46,A -85,B 0,C 180,E1 -2919.942,E2 -2919.942} C_VEL
LIN {X 0,Y 559.168,Z 379.462,A -85,B 0,C 180,E1 -2922.743,E2 -2922.743} C_VEL
LIN {X 0,Y 559.152,Z 379.462,A -85,B 0,C 180,E1 -2925.761,E2 -2925.761} C_VEL
LIN {X 0,Y 559.187,Z 379.458,A -85,B 0,C 180,E1 -2928.231,E2 -2928.231} C_VEL
LIN {X 0,Y 559.197,Z 379.598,A -85,B 0,C 180,E1 -2931.252,E2 -2931.252} C_VEL
LIN {X 0,Y 559.671,Z 384.383,A -85,B 0,C 180,E1 -2932.29,E2 -2932.29} C_VEL
LIN {X 0,Y 559.414,Z 397.721,A -85,B 0,C 180,E1 -2934.951,E2 -2934.951} C_VEL
LIN {X 0,Y 559.631,Z 414.715,A -85,B 0,C 180,E1 -2938.166,E2 -2938.166} C_VEL
LIN {X 0,Y 559.817,Z 429.625,A -85,B 0,C 180,E1 -2940.891,E2 -2940.891} C_VEL
LIN {X 0,Y 559.905,Z 446.568,A -85,B 0,C 180,E1 -2943.939,E2 -2943.939} C_VEL
LIN {X 0,Y 559.873,Z 455.052,A -85,B 0,C 180,E1 -2945.528,E2 -2945.528} C_VEL
LIN {X 0,Y 559.637,Z 468.792,A -85,B 0,C 180,E1 -2948.327,E2 -2948.327} C_VEL
LIN {X 0,Y 559.436,Z 483.739,A -85,B 0,C 180,E1 -2951.315,E2 -2951.315} C_VEL
LIN {X 0,Y 559.247,Z 497.126,A -85,B 0,C 180,E1 -2953.95,E2 -2953.95} C_VEL
LIN {X 0,Y 559.244,Z 499.881,A -85,B 0,C 180,E1 -2954.476,E2 -2954.476} C_VEL
LIN {X 0,Y 560.592,Z 507.086,A -85,B 0,C 180,E1 -2954.619,E2 -2954.619} C_VEL
LIN {X 0,Y 560.464,Z 521.057,A -85,B 0,C 180,E1 -2954.917,E2 -2954.917} C_VEL
LIN {X 0,Y 560.319,Z 535.258,A -85,B 0,C 180,E1 -2955.373,E2 -2955.373} C_VEL
LIN {X 0,Y 560.148,Z 548.082,A -85,B 0,C 180,E1 -2955.93,E2 -2955.93} C_VEL
LIN {X 0,Y 559.847,Z 561.247,A -85,B 0,C 180,E1 -2956.663,E2 -2956.663} C_VEL
LIN {X 0,Y 559.646,Z 573.132,A -85,B 0,C 180,E1 -2957.489,E2 -2957.489} C_VEL
LIN {X 0,Y 559.438,Z 584.878,A -85,B 0,C 180,E1 -2958.488,E2 -2958.488} C_VEL
LIN {X 0,Y 559.273,Z 594.701,A -85,B 0,C 180,E1 -2959.501,E2 -2959.501} C_VEL
LIN {X 0,Y 559.118,Z 603.553,A -85,B 0,C 180,E1 -2960.595,E2 -2960.595} C_VEL
LIN {X 0,Y 558.986,Z 612.032,A -85,B 0,C 180,E1 -2961.868,E2 -2961.868} C_VEL
LIN {X 0,Y 558.902,Z 618.861,A -85,B 0,C 180,E1 -2963.139,E2 -2963.139} C_VEL
LIN {X 0,Y 558.917,Z 623.565,A -85,B 0,C 180,E1 -2964.226,E2 -2964.226} C_VEL
LIN {X 0,Y 558.865,Z 628.443,A -85,B 0,C 180,E1 -2965.672,E2 -2965.672} C_VEL
LIN {X 0,Y 558.796,Z 631.832,A -85,B 0,C 180,E1 -2967.116,E2 -2967.116} C_VEL
LIN {X 0,Y 558.74,Z 633.833,A -85,B 0,C 180,E1 -2968.558,E2 -2968.558} C_VEL
LIN {X 0,Y 558.738,Z 634.5,A -85,B 0,C 180,E1 -2969.999,E2 -2969.999} C_VEL
LIN {X 0,Y 558.74,Z 633.834,A -85,B 0,C 180,E1 -2971.441,E2 -2971.441} C_VEL
LIN {X 0,Y 558.795,Z 631.833,A -85,B 0,C 180,E1 -2972.883,E2 -2972.883} C_VEL
LIN {X 0,Y 558.865,Z 628.446,A -85,B 0,C 180,E1 -2974.326,E2 -2974.326} C_VEL
LIN {X 0,Y 558.913,Z 623.572,A -85,B 0,C 180,E1 -2975.773,E2 -2975.773} C_VEL
LIN {X 0,Y 558.902,Z 618.87,A -85,B 0,C 180,E1 -2976.86,E2 -2976.86} C_VEL
LIN {X 0,Y 558.985,Z 612.042,A -85,B 0,C 180,E1 -2978.131,E2 -2978.131} C_VEL
LIN {X 0,Y 559.12,Z 603.565,A -85,B 0,C 180,E1 -2979.404,E2 -2979.404} C_VEL
LIN {X 0,Y 559.272,Z 594.715,A -85,B 0,C 180,E1 -2980.498,E2 -2980.498} C_VEL
LIN {X 0,Y 559.485,Z 584,A -85,B 0,C 180,E1 -2981.594,E2 -2981.594} C_VEL
LIN {X 0,Y 559.644,Z 573.152,A -85,B 0,C 180,E1 -2982.51,E2 -2982.51} C_VEL
LIN {X 0,Y 559.845,Z 561.269,A -85,B 0,C 180,E1 -2983.336,E2 -2983.336} C_VEL
LIN {X 0,Y 560.134,Z 548.117,A -85,B 0,C 180,E1 -2984.068,E2 -2984.068} C_VEL
LIN {X 0,Y 560.363,Z 535.32,A -85,B 0,C 180,E1 -2984.624,E2 -2984.624} C_VEL
LIN {X 0,Y 560.468,Z 521.007,A -85,B 0,C 180,E1 -2985.084,E2 -2985.084} C_VEL
LIN {X 0,Y 560.519,Z 506.632,A -85,B 0,C 180,E1 -2985.39,E2 -2985.39} C_VEL
LIN {X 0,Y 559.238,Z 499.764,A -85,B 0,C 180,E1 -2985.535,E2 -2985.535} C_VEL
LIN {X 0,Y 559.422,Z 485.66,A -85,B 0,C 180,E1 -2988.304,E2 -2988.304} C_VEL
LIN {X 0,Y 559.573,Z 472.272,A -85,B 0,C 180,E1 -2990.973,E2 -2990.973} C_VEL
LIN {X 0,Y 559.799,Z 458.885,A -85,B 0,C 180,E1 -2993.686,E2 -2993.686} C_VEL
LIN {X 0,Y 559.944,Z 446.999,A -85,B 0,C 180,E1 -2996.058,E2 -2996.058} C_VEL
LIN {X 0,Y 560.109,Z 430.775,A -85,B 0,C 180,E1 -2999.297,E2 -2999.297} C_VEL
LIN {X 0,Y 560.163,Z 417.457,A -85,B 0,C 180,E1 -3002.01,E2 -3002.01} C_VEL
LIN {X 0,Y 560.278,Z 404.38,A -85,B 0,C 180,E1 -3004.801,E2 -3004.801} C_VEL
LIN {X 0,Y 560.579,Z 392.517,A -85,B 0,C 180,E1 -3007.415,E2 -3007.415} C_VEL
LIN {X 0,Y 560.57,Z 386.397,A -85,B 0,C 180,E1 -3008.817,E2 -3008.817} C_VEL
LIN {X 0,Y 559.2,Z 379.455,A -85,B 0,C 180,E1 -3010.586,E2 -3010.586} C_VEL
LIN {X 0,Y 559.161,Z 379.457,A -85,B 0,C 180,E1 -3013.198,E2 -3013.198} C_VEL
LIN {X 0,Y 559.158,Z 379.457,A -85,B 0,C 180,E1 -3016.268,E2 -3016.268} C_VEL
LIN {X 0,Y 559.173,Z 379.454,A -85,B 0,C 180,E1 -3019.189,E2 -3019.189} C_VEL
LIN {X 0,Y 559.128,Z 379.464,A -85,B 0,C 180,E1 -3021.982,E2 -3021.982} C_VEL
LIN {X 0,Y 559.149,Z 379.455,A -85,B 0,C 180,E1 -3024.677,E2 -3024.677} C_VEL
LIN {X 0,Y 559.166,Z 379.458,A -85,B 0,C 180,E1 -3027.36,E2 -3027.36} C_VEL
LIN {X 0,Y 559.18,Z 379.455,A -85,B 0,C 180,E1 -3030.134,E2 -3030.134} C_VEL
LIN {X 0,Y 559.174,Z 379.455,A -85,B 0,C 180,E1 -3033.169,E2 -3033.169} C_VEL
LIN {X 0,Y 559.147,Z 379.463,A -85,B 0,C 180,E1 -3035.495,E2 -3035.495} C_VEL
LIN {X 0,Y 559.168,Z 379.453,A -85,B 0,C 180,E1 -3038.624,E2 -3038.624} C_VEL
LIN {X 0,Y 559.162,Z 379.455,A -85,B 0,C 180,E1 -3040.926,E2 -3040.926} C_VEL
LIN {X 0,Y 559.163,Z 379.458,A -85,B 0,C 180,E1 -3043.948,E2 -3043.948} C_VEL
LIN {X 0,Y 559.164,Z 379.455,A -85,B 0,C 180,E1 -3046.184,E2 -3046.184} C_VEL
LIN {X 0,Y 559.201,Z 379.452,A -85,B 0,C 180,E1 -3049.134,E2 -3049.134} C_VEL
LIN {X 0,Y 559.201,Z 379.451,A -85,B 0,C 180,E1 -3052.054,E2 -3052.054} C_VEL
LIN {X 0,Y 559.25,Z 379.445,A -85,B 0,C 180,E1 -3054.953,E2 -3054.953} C_VEL
LIN {X 0,Y 559.243,Z 379.448,A -85,B 0,C 180,E1 -3057.84,E2 -3057.84} C_VEL
LIN {X 0,Y 559.268,Z 379.441,A -85,B 0,C 180,E1 -3060.72,E2 -3060.72} C_VEL
LIN {X 0,Y 559.236,Z 379.446,A -85,B 0,C 180,E1 -3062.882,E2 -3062.882} C_VEL
LIN {X 0,Y 559.222,Z 379.451,A -85,B 0,C 180,E1 -3065.77,E2 -3065.77} C_VEL
LIN {X 0,Y 559.194,Z 379.45,A -85,B 0,C 180,E1 -3068.674,E2 -3068.674} C_VEL
LIN {X 0,Y 559.199,Z 379.455,A -85,B 0,C 180,E1 -3071.601,E2 -3071.601} C_VEL
LIN {X 0,Y 559.189,Z 379.451,A -85,B 0,C 180,E1 -3074.596,E2 -3074.596} C_VEL
LIN {X 0,Y 559.156,Z 379.461,A -85,B 0,C 180,E1 -3077.557,E2 -3077.557} C_VEL
LIN {X 0,Y 559.166,Z 379.456,A -85,B 0,C 180,E1 -3079.838,E2 -3079.838} C_VEL
LIN {X 0,Y 559.135,Z 379.457,A -85,B 0,C 180,E1 -3082.153,E2 -3082.153} C_VEL
LIN {X 0,Y 559.171,Z 379.461,A -85,B 0,C 180,E1 -3085.188,E2 -3085.188} C_VEL
LIN {X 0,Y 559.188,Z 379.454,A -85,B 0,C 180,E1 -3087.712,E2 -3087.712} C_VEL
LIN {X 0,Y 559.139,Z 379.458,A -85,B 0,C 180,E1 -3090.631,E2 -3090.631} C_VEL
LIN {X 0,Y 558.481,Z 379.547,A -85,B 0,C 180,E1 -3091.232,E2 -3091.232} C_VEL
LIN {X 0,Y 555.621,Z 379.902,A -85,B 0,C 180,E1 -3092.208,E2 -3092.208} C_VEL
LIN {X 0,Y 553.209,Z 380.201,A -85,B 0,C 180,E1 -3092.994,E2 -3092.994} C_VEL
LIN {X 0,Y 552.19,Z 380.326,A -85,B 0,C 180,E1 -3093.601,E2 -3093.601} C_VEL
LIN {X 0,Y 552.116,Z 380.332,A -85,B 0,C 180,E1 -3093.806,E2 -3093.806} C_VEL
LIN {X 0,Y 552.106,Z 380.336,A -85,B 0,C 180,E1 -3096.747,E2 -3096.747} C_VEL
LIN {X 0,Y 552.129,Z 380.334,A -85,B 0,C 180,E1 -3099.528,E2 -3099.528} C_VEL
LIN {X 0,Y 552.126,Z 380.331,A -85,B 0,C 180,E1 -3102.426,E2 -3102.426} C_VEL
LIN {X 0,Y 552.095,Z 380.338,A -85,B 0,C 180,E1 -3105.564,E2 -3105.564} C_VEL
LIN {X 0,Y 552.137,Z 380.332,A -85,B 0,C 180,E1 -3108.677,E2 -3108.677} C_VEL
LIN {X 0,Y 552.118,Z 380.336,A -85,B 0,C 180,E1 -3111.413,E2 -3111.413} C_VEL
LIN {X 0,Y 552.112,Z 380.332,A -85,B 0,C 180,E1 -3114.16,E2 -3114.16} C_VEL
LIN {X 0,Y 552.122,Z 380.337,A -85,B 0,C 180,E1 -3116.816,E2 -3116.816} C_VEL
LIN {X 0,Y 552.107,Z 380.337,A -85,B 0,C 180,E1 -3119.392,E2 -3119.392} C_VEL
LIN {X 0,Y 552.119,Z 380.331,A -85,B 0,C 180,E1 -3121.903,E2 -3121.903} C_VEL
LIN {X 0,Y 552.156,Z 380.331,A -85,B 0,C 180,E1 -3124.651,E2 -3124.651} C_VEL
LIN {X 0,Y 552.094,Z 380.336,A -85,B 0,C 180,E1 -3127.55,E2 -3127.55} C_VEL
LIN {X 0,Y 552.146,Z 380.33,A -85,B 0,C 180,E1 -3130.376,E2 -3130.376} C_VEL
LIN {X 0,Y 552.157,Z 380.334,A -85,B 0,C 180,E1 -3132.978,E2 -3132.978} C_VEL
LIN {X 0,Y 552.008,Z 380.352,A -85,B 0,C 180,E1 -3136.002,E2 -3136.002} C_VEL
LIN {X 0,Y 551.732,Z 380.387,A -85,B 0,C 180,E1 -3138.986,E2 -3138.986} C_VEL
LIN {X 0,Y 551.716,Z 381.399,A -85,B 0,C 180,E1 -3140.099,E2 -3140.099} C_VEL
LIN {X 0,Y 552.994,Z 390.337,A -85,B 0,C 180,E1 -3140.353,E2 -3140.353} C_VEL
LIN {X 0,Y 552.924,Z 402.814,A -85,B 0,C 180,E1 -3140.767,E2 -3140.767} C_VEL
LIN {X 0,Y 552.728,Z 414.897,A -85,B 0,C 180,E1 -3141.316,E2 -3141.316} C_VEL
LIN {X 0,Y 552.485,Z 427.121,A -85,B 0,C 180,E1 -3142.049,E2 -3142.049} C_VEL
LIN {X 0,Y 552.318,Z 437.88,A -85,B 0,C 180,E1 -3142.866,E2 -3142.866} C_VEL
LIN {X 0,Y 552.115,Z 447.657,A -85,B 0,C 180,E1 -3143.789,E2 -3143.789} C_VEL
LIN {X 0,Y 552.038,Z 457.048,A -85,B 0,C 180,E1 -3144.888,E2 -3144.888} C_VEL
LIN {X 0,Y 551.947,Z 464.566,A -85,B 0,C 180,E1 -3145.985,E2 -3145.985} C_VEL
LIN {X 0,Y 551.776,Z 470.613,A -85,B 0,C 180,E1 -3147.08,E2 -3147.08} C_VEL
LIN {X 0,Y 551.758,Z 475.411,A -85,B 0,C 180,E1 -3148.176,E2 -3148.176} C_VEL
LIN {X 0,Y 551.657,Z 479.106,A -85,B 0,C 180,E1 -3149.271,E2 -3149.271} C_VEL
LIN {X 0,Y 551.646,Z 481.009,A -85,B 0,C 180,E1 -3150.001,E2 -3150.001} C_VEL
LIN {X 0,Y 551.642,Z 482.503,A -85,B 0,C 180,E1 -3150.731,E2 -3150.731} C_VEL
LIN {X 0,Y 551.655,Z 484.205,A -85,B 0,C 180,E1 -3152.191,E2 -3152.191} C_VEL
LIN {X 0,Y 551.719,Z 484.48,A -85,B 0,C 180,E1 -3152.921,E2 -3152.921} C_VEL
LIN {X 0,Y 551.732,Z 484.361,A -85,B 0,C 180,E1 -3153.652,E2 -3153.652} C_VEL
LIN {X 0,Y 551.688,Z 482.878,A -85,B 0,C 180,E1 -3155.117,E2 -3155.117} C_VEL
LIN {X 0,Y 551.733,Z 480.016,A -85,B 0,C 180,E1 -3156.499,E2 -3156.499} C_VEL
LIN {X 0,Y 551.756,Z 476.279,A -85,B 0,C 180,E1 -3157.687,E2 -3157.687} C_VEL
LIN {X 0,Y 551.796,Z 471.666,A -85,B 0,C 180,E1 -3158.792,E2 -3158.792} C_VEL
LIN {X 0,Y 551.895,Z 464.697,A -85,B 0,C 180,E1 -3160.085,E2 -3160.085} C_VEL
LIN {X 0,Y 552.003,Z 456.881,A -85,B 0,C 180,E1 -3161.224,E2 -3161.224} C_VEL
LIN {X 0,Y 552.135,Z 447.55,A -85,B 0,C 180,E1 -3162.311,E2 -3162.311} C_VEL
LIN {X 0,Y 552.332,Z 437.674,A -85,B 0,C 180,E1 -3163.241,E2 -3163.241} C_VEL
LIN {X 0,Y 552.492,Z 426.525,A -85,B 0,C 180,E1 -3164.081,E2 -3164.081} C_VEL
LIN {X 0,Y 552.726,Z 415.646,A -85,B 0,C 180,E1 -3164.733,E2 -3164.733} C_VEL
LIN {X 0,Y 552.872,Z 403.384,A -85,B 0,C 180,E1 -3165.303,E2 -3165.303} C_VEL
LIN {X 0,Y 553.03,Z 390.258,A -85,B 0,C 180,E1 -3165.739,E2 -3165.739} C_VEL
LIN {X 0,Y 551.66,Z 381.4,A -85,B 0,C 180,E1 -3165.992,E2 -3165.992} C_VEL
LIN {X 0,Y 551.714,Z 380.39,A -85,B 0,C 180,E1 -3167.178,E2 -3167.178} C_VEL
LIN {X 0,Y 551.932,Z 380.361,A -85,B 0,C 180,E1 -3169.562,E2 -3169.562} C_VEL
LIN {X 0,Y 552.116,Z 380.334,A -85,B 0,C 180,E1 -3171.683,E2 -3171.683} C_VEL
LIN {X 0,Y 552.12,Z 380.337,A -85,B 0,C 180,E1 -3174.839,E2 -3174.839} C_VEL
LIN {X 0,Y 552.132,Z 380.334,A -85,B 0,C 180,E1 -3177.274,E2 -3177.274} C_VEL
LIN {X 0,Y 552.123,Z 380.331,A -85,B 0,C 180,E1 -3180.051,E2 -3180.051} C_VEL
LIN {X 0,Y 552.116,Z 380.341,A -85,B 0,C 180,E1 -3182.846,E2 -3182.846} C_VEL
LIN {X 0,Y 552.083,Z 380.337,A -85,B 0,C 180,E1 -3185.44,E2 -3185.44} C_VEL
LIN {X 0,Y 552.102,Z 380.332,A -85,B 0,C 180,E1 -3187.886,E2 -3187.886} C_VEL
LIN {X 0,Y 552.114,Z 380.34,A -85,B 0,C 180,E1 -3190.481,E2 -3190.481} C_VEL
LIN {X 0,Y 552.112,Z 380.332,A -85,B 0,C 180,E1 -3193.424,E2 -3193.424} C_VEL
LIN {X 0,Y 552.125,Z 380.335,A -85,B 0,C 180,E1 -3196.578,E2 -3196.578} C_VEL
LIN {X 0,Y 552.126,Z 380.329,A -85,B 0,C 180,E1 -3199.52,E2 -3199.52} C_VEL
LIN {X 0,Y 552.099,Z 380.337,A -85,B 0,C 180,E1 -3202.336,E2 -3202.336} C_VEL
LIN {X 0,Y 552.124,Z 380.33,A -85,B 0,C 180,E1 -3205.053,E2 -3205.053} C_VEL
LIN {X 0,Y 552.12,Z 380.335,A -85,B 0,C 180,E1 -3207.681,E2 -3207.681} C_VEL
LIN {X 0,Y 552.115,Z 380.327,A -85,B 0,C 180,E1 -3210.235,E2 -3210.235} C_VEL
LIN {X 0,Y 552.143,Z 380.325,A -85,B 0,C 180,E1 -3213,E2 -3213} C_VEL
LIN {X 0,Y 552.116,Z 380.333,A -85,B 0,C 180,E1 -3215.161,E2 -3215.161} C_VEL
LIN {X 0,Y 552.13,Z 380.33,A -85,B 0,C 180,E1 -3218.337,E2 -3218.337} C_VEL
LIN {X 0,Y 552.154,Z 380.327,A -85,B 0,C 180,E1 -3220.674,E2 -3220.674} C_VEL
LIN {X 0,Y 552.12,Z 380.337,A -85,B 0,C 180,E1 -3223.737,E2 -3223.737} C_VEL
LIN {X 0,Y 552.199,Z 380.325,A -85,B 0,C 180,E1 -3226.006,E2 -3226.006} C_VEL
LIN {X 0,Y 553.402,Z 385.044,A -85,B 0,C 180,E1 -3226.224,E2 -3226.224} C_VEL
LIN {X 0,Y 553.217,Z 397.657,A -85,B 0,C 180,E1 -3226.781,E2 -3226.781} C_VEL
LIN {X 0,Y 552.984,Z 407.863,A -85,B 0,C 180,E1 -3227.336,E2 -3227.336} C_VEL
LIN {X 0,Y 552.771,Z 417.802,A -85,B 0,C 180,E1 -3227.983,E2 -3227.983} C_VEL
LIN {X 0,Y 552.62,Z 427.146,A -85,B 0,C 180,E1 -3228.702,E2 -3228.702} C_VEL
LIN {X 0,Y 552.435,Z 436.57,A -85,B 0,C 180,E1 -3229.555,E2 -3229.555} C_VEL
LIN {X 0,Y 552.224,Z 445.232,A -85,B 0,C 180,E1 -3230.477,E2 -3230.477} C_VEL
LIN {X 0,Y 552.053,Z 454.017,A -85,B 0,C 180,E1 -3231.581,E2 -3231.581} C_VEL
LIN {X 0,Y 551.906,Z 462.379,A -85,B 0,C 180,E1 -3232.868,E2 -3232.868} C_VEL
LIN {X 0,Y 551.873,Z 469.08,A -85,B 0,C 180,E1 -3234.152,E2 -3234.152} C_VEL
LIN {X 0,Y 551.765,Z 473.746,A -85,B 0,C 180,E1 -3235.251,E2 -3235.251} C_VEL
LIN {X 0,Y 551.759,Z 477.494,A -85,B 0,C 180,E1 -3236.348,E2 -3236.348} C_VEL
LIN {X 0,Y 551.732,Z 479.568,A -85,B 0,C 180,E1 -3237.079,E2 -3237.079} C_VEL
LIN {X 0,Y 551.642,Z 482.501,A -85,B 0,C 180,E1 -3238.54,E2 -3238.54} C_VEL
LIN {X 0,Y 551.637,Z 483.516,A -85,B 0,C 180,E1 -3239.27,E2 -3239.27} C_VEL
LIN {X 0,Y 551.637,Z 484.443,A -85,B 0,C 180,E1 -3240.73,E2 -3240.73} C_VEL
LIN {X 0,Y 551.652,Z 484.034,A -85,B 0,C 180,E1 -3242.19,E2 -3242.19} C_VEL
LIN {X 0,Y 551.718,Z 483.406,A -85,B 0,C 180,E1 -3242.921,E2 -3242.921} C_VEL
LIN {X 0,Y 551.703,Z 480.978,A -85,B 0,C 180,E1 -3244.383,E2 -3244.383} C_VEL
LIN {X 0,Y 551.77,Z 478.264,A -85,B 0,C 180,E1 -3245.482,E2 -3245.482} C_VEL
LIN {X 0,Y 551.764,Z 474.713,A -85,B 0,C 180,E1 -3246.582,E2 -3246.582} C_VEL
LIN {X 0,Y 551.811,Z 470.247,A -85,B 0,C 180,E1 -3247.685,E2 -3247.685} C_VEL
LIN {X 0,Y 551.871,Z 464.762,A -85,B 0,C 180,E1 -3248.79,E2 -3248.79} C_VEL
LIN {X 0,Y 551.977,Z 458.16,A -85,B 0,C 180,E1 -3249.897,E2 -3249.897} C_VEL
LIN {X 0,Y 552.074,Z 450.24,A -85,B 0,C 180,E1 -3251.008,E2 -3251.008} C_VEL
LIN {X 0,Y 552.307,Z 440.74,A -85,B 0,C 180,E1 -3252.12,E2 -3252.12} C_VEL
LIN {X 0,Y 552.508,Z 430.08,A -85,B 0,C 180,E1 -3253.142,E2 -3253.142} C_VEL
LIN {X 0,Y 552.746,Z 419.564,A -85,B 0,C 180,E1 -3253.98,E2 -3253.98} C_VEL
LIN {X 0,Y 552.981,Z 409.867,A -85,B 0,C 180,E1 -3254.631,E2 -3254.631} C_VEL
LIN {X 0,Y 553.179,Z 400.408,A -85,B 0,C 180,E1 -3255.169,E2 -3255.169} C_VEL
LIN {X 0,Y 553.345,Z 388.907,A -85,B 0,C 180,E1 -3255.705,E2 -3255.705} C_VEL
LIN {X 0,Y 553.208,Z 384.383,A -85,B 0,C 180,E1 -3255.898,E2 -3255.898} C_VEL
LIN {X 0,Y 552.157,Z 380.333,A -85,B 0,C 180,E1 -3256.072,E2 -3256.072} C_VEL
LIN {X 0,Y 552.16,Z 380.333,A -85,B 0,C 180,E1 -3259.325,E2 -3259.325} C_VEL
LIN {X 0,Y 552.099,Z 380.341,A -85,B 0,C 180,E1 -3262.451,E2 -3262.451} C_VEL
LIN {X 0,Y 552.158,Z 380.335,A -85,B 0,C 180,E1 -3265.35,E2 -3265.35} C_VEL
LIN {X 0,Y 552.126,Z 380.336,A -85,B 0,C 180,E1 -3268.097,E2 -3268.097} C_VEL
LIN {X 0,Y 552.105,Z 380.339,A -85,B 0,C 180,E1 -3270.609,E2 -3270.609} C_VEL
LIN {X 0,Y 552.126,Z 380.336,A -85,B 0,C 180,E1 -3273.185,E2 -3273.185} C_VEL
LIN {X 0,Y 552.088,Z 380.341,A -85,B 0,C 180,E1 -3275.843,E2 -3275.843} C_VEL
LIN {X 0,Y 552.121,Z 380.337,A -85,B 0,C 180,E1 -3278.589,E2 -3278.589} C_VEL
LIN {X 0,Y 552.136,Z 380.337,A -85,B 0,C 180,E1 -3281.445,E2 -3281.445} C_VEL
LIN {X 0,Y 552.098,Z 380.341,A -85,B 0,C 180,E1 -3284.531,E2 -3284.531} C_VEL
LIN {X 0,Y 552.134,Z 380.338,A -85,B 0,C 180,E1 -3287.584,E2 -3287.584} C_VEL
LIN {X 0,Y 552.137,Z 380.338,A -85,B 0,C 180,E1 -3290.473,E2 -3290.473} C_VEL
LIN {X 0,Y 552.145,Z 380.394,A -85,B 0,C 180,E1 -3291.058,E2 -3291.058} C_VEL
LIN {X 0,Y 552.712,Z 384.715,A -85,B 0,C 180,E1 -3292.033,E2 -3292.033} C_VEL
LIN {X 0,Y 552.466,Z 396.728,A -85,B 0,C 180,E1 -3294.504,E2 -3294.504} C_VEL
LIN {X 0,Y 552.54,Z 413.238,A -85,B 0,C 180,E1 -3297.709,E2 -3297.709} C_VEL
LIN {X 0,Y 552.761,Z 428.106,A -85,B 0,C 180,E1 -3300.482,E2 -3300.482} C_VEL
LIN {X 0,Y 552.789,Z 443.116,A -85,B 0,C 180,E1 -3303.223,E2 -3303.223} C_VEL
LIN {X 0,Y 552.821,Z 457.315,A -85,B 0,C 180,E1 -3305.795,E2 -3305.795} C_VEL
LIN {X 0,Y 552.763,Z 464.614,A -85,B 0,C 180,E1 -3307.183,E2 -3307.183} C_VEL
LIN {X 0,Y 552.505,Z 480.287,A -85,B 0,C 180,E1 -3310.375,E2 -3310.375} C_VEL
LIN {X 0,Y 552.291,Z 495.214,A -85,B 0,C 180,E1 -3313.362,E2 -3313.362} C_VEL
LIN {X 0,Y 552.213,Z 499.88,A -85,B 0,C 180,E1 -3314.273,E2 -3314.273} C_VEL
LIN {X 0,Y 553.763,Z 508.591,A -85,B 0,C 180,E1 -3314.448,E2 -3314.448} C_VEL
LIN {X 0,Y 553.588,Z 523.083,A -85,B 0,C 180,E1 -3314.781,E2 -3314.781} C_VEL
LIN {X 0,Y 553.425,Z 536.603,A -85,B 0,C 180,E1 -3315.241,E2 -3315.241} C_VEL
LIN {X 0,Y 553.194,Z 549.864,A -85,B 0,C 180,E1 -3315.844,E2 -3315.844} C_VEL
LIN {X 0,Y 552.875,Z 562.67,A -85,B 0,C 180,E1 -3316.585,E2 -3316.585} C_VEL
LIN {X 0,Y 552.655,Z 574.303,A -85,B 0,C 180,E1 -3317.421,E2 -3317.421} C_VEL
LIN {X 0,Y 552.447,Z 585.463,A -85,B 0,C 180,E1 -3318.396,E2 -3318.396} C_VEL
LIN {X 0,Y 552.228,Z 596.327,A -85,B 0,C 180,E1 -3319.551,E2 -3319.551} C_VEL
LIN {X 0,Y 552.071,Z 604.906,A -85,B 0,C 180,E1 -3320.658,E2 -3320.658} C_VEL
LIN {X 0,Y 551.902,Z 613.114,A -85,B 0,C 180,E1 -3321.947,E2 -3321.947} C_VEL
LIN {X 0,Y 551.823,Z 618.859,A -85,B 0,C 180,E1 -3323.05,E2 -3323.05} C_VEL
LIN {X 0,Y 551.794,Z 624.958,A -85,B 0,C 180,E1 -3324.518,E2 -3324.518} C_VEL
LIN {X 0,Y 551.76,Z 628.443,A -85,B 0,C 180,E1 -3325.616,E2 -3325.616} C_VEL
LIN {X 0,Y 551.72,Z 631.833,A -85,B 0,C 180,E1 -3327.079,E2 -3327.079} C_VEL
LIN {X 0,Y 551.64,Z 633.833,A -85,B 0,C 180,E1 -3328.539,E2 -3328.539} C_VEL
LIN {X 0,Y 551.639,Z 634.5,A -85,B 0,C 180,E1 -3329.999,E2 -3329.999} C_VEL
LIN {X 0,Y 551.64,Z 633.834,A -85,B 0,C 180,E1 -3331.459,E2 -3331.459} C_VEL
LIN {X 0,Y 551.719,Z 631.834,A -85,B 0,C 180,E1 -3332.92,E2 -3332.92} C_VEL
LIN {X 0,Y 551.759,Z 628.446,A -85,B 0,C 180,E1 -3334.382,E2 -3334.382} C_VEL
LIN {X 0,Y 551.822,Z 623.572,A -85,B 0,C 180,E1 -3335.847,E2 -3335.847} C_VEL
LIN {X 0,Y 551.832,Z 617.058,A -85,B 0,C 180,E1 -3337.316,E2 -3337.316} C_VEL
LIN {X 0,Y 551.962,Z 609.806,A -85,B 0,C 180,E1 -3338.603,E2 -3338.603} C_VEL
LIN {X 0,Y 552.115,Z 600.83,A -85,B 0,C 180,E1 -3339.894,E2 -3339.894} C_VEL
LIN {X 0,Y 552.345,Z 591.401,A -85,B 0,C 180,E1 -3341.002,E2 -3341.002} C_VEL
LIN {X 0,Y 552.538,Z 580.964,A -85,B 0,C 180,E1 -3342.021,E2 -3342.021} C_VEL
LIN {X 0,Y 552.762,Z 569.446,A -85,B 0,C 180,E1 -3342.948,E2 -3342.948} C_VEL
LIN {X 0,Y 553.019,Z 556.656,A -85,B 0,C 180,E1 -3343.784,E2 -3343.784} C_VEL
LIN {X 0,Y 553.281,Z 544.176,A -85,B 0,C 180,E1 -3344.434,E2 -3344.434} C_VEL
LIN {X 0,Y 553.53,Z 531.058,A -85,B 0,C 180,E1 -3344.964,E2 -3344.964} C_VEL
LIN {X 0,Y 553.644,Z 517.469,A -85,B 0,C 180,E1 -3345.366,E2 -3345.366} C_VEL
LIN {X 0,Y 553.649,Z 507.573,A -85,B 0,C 180,E1 -3345.571,E2 -3345.571} C_VEL
LIN {X 0,Y 552.223,Z 499.764,A -85,B 0,C 180,E1 -3345.737,E2 -3345.737} C_VEL
LIN {X 0,Y 552.428,Z 485.66,A -85,B 0,C 180,E1 -3348.544,E2 -3348.544} C_VEL
LIN {X 0,Y 552.656,Z 470.36,A -85,B 0,C 180,E1 -3351.64,E2 -3351.64} C_VEL
LIN {X 0,Y 552.806,Z 458.549,A -85,B 0,C 180,E1 -3354.004,E2 -3354.004} C_VEL
LIN {X 0,Y 552.931,Z 446.374,A -85,B 0,C 180,E1 -3356.414,E2 -3356.414} C_VEL
LIN {X 0,Y 553.13,Z 431.214,A -85,B 0,C 180,E1 -3359.494,E2 -3359.494} C_VEL
LIN {X 0,Y 553.242,Z 417.982,A -85,B 0,C 180,E1 -3362.244,E2 -3362.244} C_VEL
LIN {X 0,Y 553.408,Z 404.116,A -85,B 0,C 180,E1 -3365.249,E2 -3365.249} C_VEL
LIN {X 0,Y 553.743,Z 392.678,A -85,B 0,C 180,E1 -3367.817,E2 -3367.817} C_VEL
LIN {X 0,Y 553.732,Z 388.338,A -85,B 0,C 180,E1 -3368.829,E2 -3368.829} C_VEL
LIN {X 0,Y 552.145,Z 380.334,A -85,B 0,C 180,E1 -3370.897,E2 -3370.897} C_VEL
LIN {X 0,Y 552.108,Z 380.339,A -85,B 0,C 180,E1 -3373.483,E2 -3373.483} C_VEL
LIN {X 0,Y 552.116,Z 380.332,A -85,B 0,C 180,E1 -3376.577,E2 -3376.577} C_VEL
LIN {X 0,Y 552.137,Z 380.335,A -85,B 0,C 180,E1 -3379.521,E2 -3379.521} C_VEL
LIN {X 0,Y 552.086,Z 380.337,A -85,B 0,C 180,E1 -3382.336,E2 -3382.336} C_VEL
LIN {X 0,Y 552.121,Z 380.332,A -85,B 0,C 180,E1 -3385.054,E2 -3385.054} C_VEL
LIN {X 0,Y 552.12,Z 380.339,A -85,B 0,C 180,E1 -3387.682,E2 -3387.682} C_VEL
LIN {X 0,Y 552.136,Z 380.331,A -85,B 0,C 180,E1 -3390.237,E2 -3390.237} C_VEL
LIN {X 0,Y 552.138,Z 380.33,A -85,B 0,C 180,E1 -3392.997,E2 -3392.997} C_VEL
LIN {X 0,Y 552.103,Z 380.336,A -85,B 0,C 180,E1 -3395.161,E2 -3395.161} C_VEL
LIN {X 0,Y 552.087,Z 380.344,A -85,B 0,C 180,E1 -3397.549,E2 -3397.549} C_VEL
LIN {X 0,Y 552.139,Z 380.329,A -85,B 0,C 180,E1 -3400.373,E2 -3400.373} C_VEL
LIN {X 0,Y 552.149,Z 380.329,A -85,B 0,C 180,E1 -3402.977,E2 -3402.977} C_VEL
LIN {X 0,Y 552.127,Z 380.334,A -85,B 0,C 180,E1 -3406.004,E2 -3406.004} C_VEL
LIN {X 0,Y 552.168,Z 380.327,A -85,B 0,C 180,E1 -3408.994,E2 -3408.994} C_VEL
LIN {X 0,Y 552.154,Z 380.33,A -85,B 0,C 180,E1 -3411.952,E2 -3411.952} C_VEL
LIN {X 0,Y 552.224,Z 380.32,A -85,B 0,C 180,E1 -3414.889,E2 -3414.889} C_VEL
LIN {X 0,Y 552.215,Z 380.324,A -85,B 0,C 180,E1 -3417.812,E2 -3417.812} C_VEL
LIN {X 0,Y 552.238,Z 380.317,A -85,B 0,C 180,E1 -3420.729,E2 -3420.729} C_VEL
LIN {X 0,Y 552.202,Z 380.323,A -85,B 0,C 180,E1 -3422.918,E2 -3422.918} C_VEL
LIN {X 0,Y 552.191,Z 380.326,A -85,B 0,C 180,E1 -3425.844,E2 -3425.844} C_VEL
LIN {X 0,Y 552.162,Z 380.327,A -85,B 0,C 180,E1 -3428.786,E2 -3428.786} C_VEL
LIN {X 0,Y 552.155,Z 380.331,A -85,B 0,C 180,E1 -3431.751,E2 -3431.751} C_VEL
LIN {X 0,Y 552.127,Z 380.332,A -85,B 0,C 180,E1 -3434.749,E2 -3434.749} C_VEL
LIN {X 0,Y 552.107,Z 380.336,A -85,B 0,C 180,E1 -3437.789,E2 -3437.789} C_VEL
LIN {X 0,Y 552.125,Z 380.331,A -85,B 0,C 180,E1 -3440.102,E2 -3440.102} C_VEL
LIN {X 0,Y 552.088,Z 380.335,A -85,B 0,C 180,E1 -3442.451,E2 -3442.451} C_VEL
LIN {X 0,Y 552.148,Z 380.335,A -85,B 0,C 180,E1 -3445.352,E2 -3445.352} C_VEL
LIN {X 0,Y 552.119,Z 380.331,A -85,B 0,C 180,E1 -3448.098,E2 -3448.098} C_VEL
LIN {X 0,Y 552.1,Z 380.335,A -85,B 0,C 180,E1 -3450.626,E2 -3450.626} C_VEL
LIN {X 0,Y 552.122,Z 380.339,A -85,B 0,C 180,E1 -3453.186,E2 -3453.186} C_VEL
LIN {X 0,Y 552.116,Z 380.332,A -85,B 0,C 180,E1 -3453.806,E2 -3453.806} C_VEL
LIN {X 0,Y 551.481,Z 380.412,A -85,B 0,C 180,E1 -3454.415,E2 -3454.415} C_VEL
LIN {X 0,Y 548.655,Z 380.769,A -85,B 0,C 180,E1 -3455.403,E2 -3455.403} C_VEL
LIN {X 0,Y 546.23,Z 381.071,A -85,B 0,C 180,E1 -3456.198,E2 -3456.198} C_VEL
LIN {X 0,Y 545.16,Z 381.204,A -85,B 0,C 180,E1 -3456.812,E2 -3456.812} C_VEL
LIN {X 0,Y 545.058,Z 381.216,A -85,B 0,C 180,E1 -3457.02,E2 -3457.02} C_VEL
LIN {X 0,Y 545.069,Z 381.21,A -85,B 0,C 180,E1 -3460.143,E2 -3460.143} C_VEL
LIN {X 0,Y 545.083,Z 381.215,A -85,B 0,C 180,E1 -3463.107,E2 -3463.107} C_VEL
LIN {X 0,Y 545.063,Z 381.211,A -85,B 0,C 180,E1 -3466.225,E2 -3466.225} C_VEL
LIN {X 0,Y 545.098,Z 381.212,A -85,B 0,C 180,E1 -3468.889,E2 -3468.889} C_VEL
LIN {X 0,Y 545.052,Z 381.213,A -85,B 0,C 180,E1 -3471.764,E2 -3471.764} C_VEL
LIN {X 0,Y 545.064,Z 381.212,A -85,B 0,C 180,E1 -3474.535,E2 -3474.535} C_VEL
LIN {X 0,Y 545.08,Z 381.214,A -85,B 0,C 180,E1 -3477.214,E2 -3477.214} C_VEL
LIN {X 0,Y 545.066,Z 381.211,A -85,B 0,C 180,E1 -3479.812,E2 -3479.812} C_VEL
LIN {X 0,Y 545.089,Z 381.208,A -85,B 0,C 180,E1 -3482.345,E2 -3482.345} C_VEL
LIN {X 0,Y 545.118,Z 381.21,A -85,B 0,C 180,E1 -3484.822,E2 -3484.822} C_VEL
LIN {X 0,Y 545.04,Z 381.219,A -85,B 0,C 180,E1 -3487.243,E2 -3487.243} C_VEL
LIN {X 0,Y 545.118,Z 381.206,A -85,B 0,C 180,E1 -3490.416,E2 -3490.416} C_VEL
LIN {X 0,Y 545.069,Z 381.211,A -85,B 0,C 180,E1 -3493.522,E2 -3493.522} C_VEL
LIN {X 0,Y 544.985,Z 381.226,A -85,B 0,C 180,E1 -3495.818,E2 -3495.818} C_VEL
LIN {X 0,Y 544.714,Z 381.263,A -85,B 0,C 180,E1 -3498.842,E2 -3498.842} C_VEL
LIN {X 0,Y 544.622,Z 381.392,A -85,B 0,C 180,E1 -3499.921,E2 -3499.921} C_VEL
LIN {X 0,Y 546.076,Z 390.918,A -85,B 0,C 180,E1 -3500.206,E2 -3500.206} C_VEL
LIN {X 0,Y 545.977,Z 403.836,A -85,B 0,C 180,E1 -3500.648,E2 -3500.648} C_VEL
LIN {X 0,Y 545.767,Z 415.626,A -85,B 0,C 180,E1 -3501.205,E2 -3501.205} C_VEL
LIN {X 0,Y 545.497,Z 427.704,A -85,B 0,C 180,E1 -3501.947,E2 -3501.947} C_VEL
LIN {X 0,Y 545.291,Z 438.53,A -85,B 0,C 180,E1 -3502.791,E2 -3502.791} C_VEL
LIN {X 0,Y 545.063,Z 448.027,A -85,B 0,C 180,E1 -3503.709,E2 -3503.709} C_VEL
LIN {X 0,Y 544.972,Z 457.351,A -85,B 0,C 180,E1 -3504.822,E2 -3504.822} C_VEL
LIN {X 0,Y 544.88,Z 464.802,A -85,B 0,C 180,E1 -3505.933,E2 -3505.933} C_VEL
LIN {X 0,Y 544.706,Z 470.802,A -85,B 0,C 180,E1 -3507.043,E2 -3507.043} C_VEL
LIN {X 0,Y 544.679,Z 475.56,A -85,B 0,C 180,E1 -3508.152,E2 -3508.152} C_VEL
LIN {X 0,Y 544.559,Z 479.217,A -85,B 0,C 180,E1 -3509.261,E2 -3509.261} C_VEL
LIN {X 0,Y 544.547,Z 481.103,A -85,B 0,C 180,E1 -3510.001,E2 -3510.001} C_VEL
LIN {X 0,Y 544.543,Z 482.568,A -85,B 0,C 180,E1 -3510.74,E2 -3510.74} C_VEL
LIN {X 0,Y 544.57,Z 484.23,A -85,B 0,C 180,E1 -3512.22,E2 -3512.22} C_VEL
LIN {X 0,Y 544.645,Z 484.488,A -85,B 0,C 180,E1 -3512.959,E2 -3512.959} C_VEL
LIN {X 0,Y 544.646,Z 484.338,A -85,B 0,C 180,E1 -3513.7,E2 -3513.7} C_VEL
LIN {X 0,Y 544.61,Z 482.818,A -85,B 0,C 180,E1 -3515.183,E2 -3515.183} C_VEL
LIN {X 0,Y 544.644,Z 480.166,A -85,B 0,C 180,E1 -3516.484,E2 -3516.484} C_VEL
LIN {X 0,Y 544.672,Z 476.127,A -85,B 0,C 180,E1 -3517.787,E2 -3517.787} C_VEL
LIN {X 0,Y 544.733,Z 471.473,A -85,B 0,C 180,E1 -3518.907,E2 -3518.907} C_VEL
LIN {X 0,Y 544.843,Z 464.456,A -85,B 0,C 180,E1 -3520.217,E2 -3520.217} C_VEL
LIN {X 0,Y 544.953,Z 457.234,A -85,B 0,C 180,E1 -3521.285,E2 -3521.285} C_VEL
LIN {X 0,Y 545.078,Z 448.922,A -85,B 0,C 180,E1 -3522.284,E2 -3522.284} C_VEL
LIN {X 0,Y 545.26,Z 439.342,A -85,B 0,C 180,E1 -3523.226,E2 -3523.226} C_VEL
LIN {X 0,Y 545.472,Z 428.694,A -85,B 0,C 180,E1 -3524.076,E2 -3524.076} C_VEL
LIN {X 0,Y 545.749,Z 416.616,A -85,B 0,C 180,E1 -3524.83,E2 -3524.83} C_VEL
LIN {X 0,Y 545.922,Z 404.333,A -85,B 0,C 180,E1 -3525.422,E2 -3525.422} C_VEL
LIN {X 0,Y 546.107,Z 391.333,A -85,B 0,C 180,E1 -3525.872,E2 -3525.872} C_VEL
LIN {X 0,Y 544.565,Z 381.406,A -85,B 0,C 180,E1 -3526.158,E2 -3526.158} C_VEL
LIN {X 0,Y 544.817,Z 381.248,A -85,B 0,C 180,E1 -3528.814,E2 -3528.814} C_VEL
LIN {X 0,Y 545.071,Z 381.21,A -85,B 0,C 180,E1 -3531.82,E2 -3531.82} C_VEL
LIN {X 0,Y 545.055,Z 381.212,A -85,B 0,C 180,E1 -3534.37,E2 -3534.37} C_VEL
LIN {X 0,Y 545.09,Z 381.213,A -85,B 0,C 180,E1 -3537.172,E2 -3537.172} C_VEL
LIN {X 0,Y 545.071,Z 381.213,A -85,B 0,C 180,E1 -3539.339,E2 -3539.339} C_VEL
LIN {X 0,Y 545.06,Z 381.211,A -85,B 0,C 180,E1 -3541.915,E2 -3541.915} C_VEL
LIN {X 0,Y 545.066,Z 381.217,A -85,B 0,C 180,E1 -3544.565,E2 -3544.565} C_VEL
LIN {X 0,Y 545.041,Z 381.212,A -85,B 0,C 180,E1 -3547.304,E2 -3547.304} C_VEL
LIN {X 0,Y 545.071,Z 381.211,A -85,B 0,C 180,E1 -3550.143,E2 -3550.143} C_VEL
LIN {X 0,Y 545.084,Z 381.208,A -85,B 0,C 180,E1 -3553.107,E2 -3553.107} C_VEL
LIN {X 0,Y 545.07,Z 381.215,A -85,B 0,C 180,E1 -3556.224,E2 -3556.224} C_VEL
LIN {X 0,Y 545.103,Z 381.204,A -85,B 0,C 180,E1 -3558.887,E2 -3558.887} C_VEL
LIN {X 0,Y 545.059,Z 381.207,A -85,B 0,C 180,E1 -3561.763,E2 -3561.763} C_VEL
LIN {X 0,Y 545.061,Z 381.213,A -85,B 0,C 180,E1 -3564.533,E2 -3564.533} C_VEL
LIN {X 0,Y 545.073,Z 381.208,A -85,B 0,C 180,E1 -3567.211,E2 -3567.211} C_VEL
LIN {X 0,Y 545.067,Z 381.209,A -85,B 0,C 180,E1 -3569.81,E2 -3569.81} C_VEL
LIN {X 0,Y 545.093,Z 381.205,A -85,B 0,C 180,E1 -3572.344,E2 -3572.344} C_VEL
LIN {X 0,Y 545.121,Z 381.202,A -85,B 0,C 180,E1 -3574.82,E2 -3574.82} C_VEL
LIN {X 0,Y 545.04,Z 381.216,A -85,B 0,C 180,E1 -3577.242,E2 -3577.242} C_VEL
LIN {X 0,Y 545.12,Z 381.203,A -85,B 0,C 180,E1 -3580.415,E2 -3580.415} C_VEL
LIN {X 0,Y 545.077,Z 381.217,A -85,B 0,C 180,E1 -3583.521,E2 -3583.521} C_VEL
LIN {X 0,Y 545.151,Z 381.296,A -85,B 0,C 180,E1 -3585.857,E2 -3585.857} C_VEL
LIN {X 0,Y 546.525,Z 386.476,A -85,B 0,C 180,E1 -3586.095,E2 -3586.095} C_VEL
LIN {X 0,Y 546.325,Z 397.908,A -85,B 0,C 180,E1 -3586.611,E2 -3586.611} C_VEL
LIN {X 0,Y 546.07,Z 408.073,A -85,B 0,C 180,E1 -3587.173,E2 -3587.173} C_VEL
LIN {X 0,Y 545.827,Z 417.982,A -85,B 0,C 180,E1 -3587.828,E2 -3587.828} C_VEL
LIN {X 0,Y 545.645,Z 427.61,A -85,B 0,C 180,E1 -3588.583,E2 -3588.583} C_VEL
LIN {X 0,Y 545.429,Z 436.7,A -85,B 0,C 180,E1 -3589.419,E2 -3589.419} C_VEL
LIN {X 0,Y 545.205,Z 445.345,A -85,B 0,C 180,E1 -3590.353,E2 -3590.353} C_VEL
LIN {X 0,Y 545.022,Z 454.117,A -85,B 0,C 180,E1 -3591.472,E2 -3591.472} C_VEL
LIN {X 0,Y 544.835,Z 462.447,A -85,B 0,C 180,E1 -3592.775,E2 -3592.775} C_VEL
LIN {X 0,Y 544.786,Z 469.135,A -85,B 0,C 180,E1 -3594.076,E2 -3594.076} C_VEL
LIN {X 0,Y 544.665,Z 473.79,A -85,B 0,C 180,E1 -3595.189,E2 -3595.189} C_VEL
LIN {X 0,Y 544.678,Z 477.528,A -85,B 0,C 180,E1 -3596.301,E2 -3596.301} C_VEL
LIN {X 0,Y 544.661,Z 479.602,A -85,B 0,C 180,E1 -3597.041,E2 -3597.041} C_VEL
LIN {X 0,Y 544.543,Z 482.515,A -85,B 0,C 180,E1 -3598.521,E2 -3598.521} C_VEL
LIN {X 0,Y 544.538,Z 483.533,A -85,B 0,C 180,E1 -3599.26,E2 -3599.26} C_VEL
LIN {X 0,Y 544.537,Z 484.436,A -85,B 0,C 180,E1 -3600.739,E2 -3600.739} C_VEL
LIN {X 0,Y 544.544,Z 484.427,A -85,B 0,C 180,E1 -3601.479,E2 -3601.479} C_VEL
LIN {X 0,Y 544.645,Z 483.387,A -85,B 0,C 180,E1 -3602.958,E2 -3602.958} C_VEL
LIN {X 0,Y 544.601,Z 480.941,A -85,B 0,C 180,E1 -3604.441,E2 -3604.441} C_VEL
LIN {X 0,Y 544.696,Z 478.218,A -85,B 0,C 180,E1 -3605.553,E2 -3605.553} C_VEL
LIN {X 0,Y 544.727,Z 473.272,A -85,B 0,C 180,E1 -3607.04,E2 -3607.04} C_VEL
LIN {X 0,Y 544.782,Z 466.706,A -85,B 0,C 180,E1 -3608.532,E2 -3608.532} C_VEL
LIN {X 0,Y 544.927,Z 459.265,A -85,B 0,C 180,E1 -3609.839,E2 -3609.839} C_VEL
LIN {X 0,Y 545.054,Z 451.534,A -85,B 0,C 180,E1 -3610.964,E2 -3610.964} C_VEL
LIN {X 0,Y 545.219,Z 443.911,A -85,B 0,C 180,E1 -3611.902,E2 -3611.902} C_VEL
LIN {X 0,Y 545.434,Z 434.974,A -85,B 0,C 180,E1 -3612.842,E2 -3612.842} C_VEL
LIN {X 0,Y 545.708,Z 424.37,A -85,B 0,C 180,E1 -3613.783,E2 -3613.783} C_VEL
LIN {X 0,Y 546.013,Z 411.155,A -85,B 0,C 180,E1 -3614.727,E2 -3614.727} C_VEL
LIN {X 0,Y 546.272,Z 400.625,A -85,B 0,C 180,E1 -3615.339,E2 -3615.339} C_VEL
LIN {X 0,Y 546.471,Z 389.687,A -85,B 0,C 180,E1 -3615.86,E2 -3615.86} C_VEL
LIN {X 0,Y 546.447,Z 386.308,A -85,B 0,C 180,E1 -3616.004,E2 -3616.004} C_VEL
LIN {X 0,Y 545.088,Z 381.215,A -85,B 0,C 180,E1 -3616.238,E2 -3616.238} C_VEL
LIN {X 0,Y 545.087,Z 381.214,A -85,B 0,C 180,E1 -3618.804,E2 -3618.804} C_VEL
LIN {X 0,Y 545.069,Z 381.216,A -85,B 0,C 180,E1 -3621.163,E2 -3621.163} C_VEL
LIN {X 0,Y 545.056,Z 381.219,A -85,B 0,C 180,E1 -3624.369,E2 -3624.369} C_VEL
LIN {X 0,Y 545.098,Z 381.211,A -85,B 0,C 180,E1 -3627.174,E2 -3627.174} C_VEL
LIN {X 0,Y 545.067,Z 381.216,A -85,B 0,C 180,E1 -3629.338,E2 -3629.338} C_VEL
LIN {X 0,Y 545.062,Z 381.216,A -85,B 0,C 180,E1 -3631.914,E2 -3631.914} C_VEL
LIN {X 0,Y 545.065,Z 381.215,A -85,B 0,C 180,E1 -3634.564,E2 -3634.564} C_VEL
LIN {X 0,Y 545.039,Z 381.219,A -85,B 0,C 180,E1 -3637.304,E2 -3637.304} C_VEL
LIN {X 0,Y 545.069,Z 381.217,A -85,B 0,C 180,E1 -3640.142,E2 -3640.142} C_VEL
LIN {X 0,Y 545.082,Z 381.214,A -85,B 0,C 180,E1 -3643.106,E2 -3643.106} C_VEL
LIN {X 0,Y 545.052,Z 381.219,A -85,B 0,C 180,E1 -3646.226,E2 -3646.226} C_VEL
LIN {X 0,Y 545.089,Z 381.216,A -85,B 0,C 180,E1 -3648.886,E2 -3648.886} C_VEL
LIN {X 0,Y 545.103,Z 381.331,A -85,B 0,C 180,E1 -3650.879,E2 -3650.879} C_VEL
LIN {X 0,Y 545.761,Z 386.398,A -85,B 0,C 180,E1 -3652.055,E2 -3652.055} C_VEL
LIN {X 0,Y 545.42,Z 399.445,A -85,B 0,C 180,E1 -3654.786,E2 -3654.786} C_VEL
LIN {X 0,Y 545.536,Z 415.217,A -85,B 0,C 180,E1 -3657.898,E2 -3657.898} C_VEL
LIN {X 0,Y 545.709,Z 430.016,A -85,B 0,C 180,E1 -3660.699,E2 -3660.699} C_VEL
LIN {X 0,Y 545.749,Z 446.929,A -85,B 0,C 180,E1 -3663.828,E2 -3663.828} C_VEL
LIN {X 0,Y 545.718,Z 463.556,A -85,B 0,C 180,E1 -3666.871,E2 -3666.871} C_VEL
LIN {X 0,Y 545.617,Z 474.169,A -85,B 0,C 180,E1 -3668.858,E2 -3668.858} C_VEL
LIN {X 0,Y 545.38,Z 487.564,A -85,B 0,C 180,E1 -3671.595,E2 -3671.595} C_VEL
LIN {X 0,Y 545.166,Z 499.756,A -85,B 0,C 180,E1 -3674.052,E2 -3674.052} C_VEL
LIN {X 0,Y 546.926,Z 509.851,A -85,B 0,C 180,E1 -3674.272,E2 -3674.272} C_VEL
LIN {X 0,Y 546.731,Z 523.545,A -85,B 0,C 180,E1 -3674.6,E2 -3674.6} C_VEL
LIN {X 0,Y 546.521,Z 537.682,A -85,B 0,C 180,E1 -3675.096,E2 -3675.096} C_VEL
LIN {X 0,Y 546.307,Z 549.862,A -85,B 0,C 180,E1 -3675.661,E2 -3675.661} C_VEL
LIN {X 0,Y 545.959,Z 562.668,A -85,B 0,C 180,E1 -3676.412,E2 -3676.412} C_VEL
LIN {X 0,Y 545.707,Z 574.301,A -85,B 0,C 180,E1 -3677.258,E2 -3677.258} C_VEL
LIN {X 0,Y 545.455,Z 585.079,A -85,B 0,C 180,E1 -3678.208,E2 -3678.208} C_VEL
LIN {X 0,Y 545.232,Z 594.701,A -85,B 0,C 180,E1 -3679.227,E2 -3679.227} C_VEL
LIN {X 0,Y 545.024,Z 603.552,A -85,B 0,C 180,E1 -3680.349,E2 -3680.349} C_VEL
LIN {X 0,Y 544.873,Z 612.031,A -85,B 0,C 180,E1 -3681.656,E2 -3681.656} C_VEL
LIN {X 0,Y 544.736,Z 618.859,A -85,B 0,C 180,E1 -3682.959,E2 -3682.959} C_VEL
LIN {X 0,Y 544.731,Z 623.565,A -85,B 0,C 180,E1 -3684.075,E2 -3684.075} C_VEL
LIN {X 0,Y 544.654,Z 628.444,A -85,B 0,C 180,E1 -3685.559,E2 -3685.559} C_VEL
LIN {X 0,Y 544.647,Z 631.833,A -85,B 0,C 180,E1 -3687.041,E2 -3687.041} C_VEL
LIN {X 0,Y 544.541,Z 633.834,A -85,B 0,C 180,E1 -3688.52,E2 -3688.52} C_VEL
LIN {X 0,Y 544.539,Z 634.5,A -85,B 0,C 180,E1 -3689.999,E2 -3689.999} C_VEL
LIN {X 0,Y 544.541,Z 633.835,A -85,B 0,C 180,E1 -3691.478,E2 -3691.478} C_VEL
LIN {X 0,Y 544.646,Z 631.834,A -85,B 0,C 180,E1 -3692.958,E2 -3692.958} C_VEL
LIN {X 0,Y 544.654,Z 628.446,A -85,B 0,C 180,E1 -3694.44,E2 -3694.44} C_VEL
LIN {X 0,Y 544.735,Z 623.572,A -85,B 0,C 180,E1 -3695.923,E2 -3695.923} C_VEL
LIN {X 0,Y 544.782,Z 617.058,A -85,B 0,C 180,E1 -3697.411,E2 -3697.411} C_VEL
LIN {X 0,Y 544.909,Z 609.807,A -85,B 0,C 180,E1 -3698.716,E2 -3698.716} C_VEL
LIN {X 0,Y 545.081,Z 600.83,A -85,B 0,C 180,E1 -3700.023,E2 -3700.023} C_VEL
LIN {X 0,Y 545.348,Z 591.401,A -85,B 0,C 180,E1 -3701.145,E2 -3701.145} C_VEL
LIN {X 0,Y 545.544,Z 580.965,A -85,B 0,C 180,E1 -3702.177,E2 -3702.177} C_VEL
LIN {X 0,Y 545.822,Z 569.444,A -85,B 0,C 180,E1 -3703.116,E2 -3703.116} C_VEL
LIN {X 0,Y 546.119,Z 556.655,A -85,B 0,C 180,E1 -3703.962,E2 -3703.962} C_VEL
LIN {X 0,Y 546.388,Z 544.174,A -85,B 0,C 180,E1 -3704.62,E2 -3704.62} C_VEL
LIN {X 0,Y 546.671,Z 531.849,A -85,B 0,C 180,E1 -3705.127,E2 -3705.127} C_VEL
LIN {X 0,Y 546.793,Z 517.792,A -85,B 0,C 180,E1 -3705.555,E2 -3705.555} C_VEL
LIN {X 0,Y 546.772,Z 508.324,A -85,B 0,C 180,E1 -3705.76,E2 -3705.76} C_VEL
LIN {X 0,Y 545.163,Z 499.764,A -85,B 0,C 180,E1 -3705.946,E2 -3705.946} C_VEL
LIN {X 0,Y 545.396,Z 487.572,A -85,B 0,C 180,E1 -3708.403,E2 -3708.403} C_VEL
LIN {X 0,Y 545.62,Z 474.177,A -85,B 0,C 180,E1 -3711.14,E2 -3711.14} C_VEL
LIN {X 0,Y 545.771,Z 460.023,A -85,B 0,C 180,E1 -3713.896,E2 -3713.896} C_VEL
LIN {X 0,Y 545.926,Z 446.754,A -85,B 0,C 180,E1 -3716.573,E2 -3716.573} C_VEL
LIN {X 0,Y 546.151,Z 431.589,A -85,B 0,C 180,E1 -3719.697,E2 -3719.697} C_VEL
LIN {X 0,Y 546.344,Z 417.447,A -85,B 0,C 180,E1 -3722.701,E2 -3722.701} C_VEL
LIN {X 0,Y 546.666,Z 401.433,A -85,B 0,C 180,E1 -3726.254,E2 -3726.254} C_VEL
LIN {X 0,Y 546.925,Z 391.045,A -85,B 0,C 180,E1 -3728.654,E2 -3728.654} C_VEL
LIN {X 0,Y 545.583,Z 383.608,A -85,B 0,C 180,E1 -3730.534,E2 -3730.534} C_VEL
LIN {X 0,Y 545.095,Z 381.213,A -85,B 0,C 180,E1 -3731.212,E2 -3731.212} C_VEL
LIN {X 0,Y 545.052,Z 381.218,A -85,B 0,C 180,E1 -3734.128,E2 -3734.128} C_VEL
LIN {X 0,Y 545.082,Z 381.208,A -85,B 0,C 180,E1 -3736.894,E2 -3736.894} C_VEL
LIN {X 0,Y 545.105,Z 381.211,A -85,B 0,C 180,E1 -3739.522,E2 -3739.522} C_VEL
LIN {X 0,Y 545.045,Z 381.22,A -85,B 0,C 180,E1 -3741.863,E2 -3741.863} C_VEL
LIN {X 0,Y 545.056,Z 381.212,A -85,B 0,C 180,E1 -3744.533,E2 -3744.533} C_VEL
LIN {X 0,Y 545.074,Z 381.212,A -85,B 0,C 180,E1 -3747.212,E2 -3747.212} C_VEL
LIN {X 0,Y 545.092,Z 381.213,A -85,B 0,C 180,E1 -3749.812,E2 -3749.812} C_VEL
LIN {X 0,Y 545.093,Z 381.207,A -85,B 0,C 180,E1 -3752.824,E2 -3752.824} C_VEL
LIN {X 0,Y 545.043,Z 381.22,A -85,B 0,C 180,E1 -3755.631,E2 -3755.631} C_VEL
LIN {X 0,Y 545.059,Z 381.211,A -85,B 0,C 180,E1 -3758.837,E2 -3758.837} C_VEL
LIN {X 0,Y 545.075,Z 381.212,A -85,B 0,C 180,E1 -3761.196,E2 -3761.196} C_VEL
LIN {X 0,Y 545.069,Z 381.217,A -85,B 0,C 180,E1 -3763.521,E2 -3763.521} C_VEL
LIN {X 0,Y 545.085,Z 381.213,A -85,B 0,C 180,E1 -3765.82,E2 -3765.82} C_VEL
LIN {X 0,Y 545.122,Z 381.204,A -85,B 0,C 180,E1 -3768.85,E2 -3768.85} C_VEL
LIN {X 0,Y 545.124,Z 381.207,A -85,B 0,C 180,E1 -3771.847,E2 -3771.847} C_VEL
LIN {X 0,Y 545.199,Z 381.194,A -85,B 0,C 180,E1 -3774.823,E2 -3774.823} C_VEL
LIN {X 0,Y 545.186,Z 381.2,A -85,B 0,C 180,E1 -3777.784,E2 -3777.784} C_VEL
LIN {X 0,Y 545.207,Z 381.193,A -85,B 0,C 180,E1 -3780.739,E2 -3780.739} C_VEL
LIN {X 0,Y 545.168,Z 381.2,A -85,B 0,C 180,E1 -3782.956,E2 -3782.956} C_VEL
LIN {X 0,Y 545.163,Z 381.201,A -85,B 0,C 180,E1 -3785.92,E2 -3785.92} C_VEL
LIN {X 0,Y 545.119,Z 381.206,A -85,B 0,C 180,E1 -3788.9,E2 -3788.9} C_VEL
LIN {X 0,Y 545.126,Z 381.205,A -85,B 0,C 180,E1 -3791.905,E2 -3791.905} C_VEL
LIN {X 0,Y 545.076,Z 381.212,A -85,B 0,C 180,E1 -3794.944,E2 -3794.944} C_VEL
LIN {X 0,Y 545.075,Z 381.21,A -85,B 0,C 180,E1 -3798.026,E2 -3798.026} C_VEL
LIN {X 0,Y 545.09,Z 381.207,A -85,B 0,C 180,E1 -3800.373,E2 -3800.373} C_VEL
LIN {X 0,Y 545.083,Z 381.214,A -85,B 0,C 180,E1 -3803.56,E2 -3803.56} C_VEL
LIN {X 0,Y 545.081,Z 381.209,A -85,B 0,C 180,E1 -3806.001,E2 -3806.001} C_VEL
LIN {X 0,Y 545.083,Z 381.21,A -85,B 0,C 180,E1 -3808.75,E2 -3808.75} C_VEL
LIN {X 0,Y 545.071,Z 381.213,A -85,B 0,C 180,E1 -3811.683,E2 -3811.683} C_VEL
LIN {X 0,Y 545.077,Z 381.21,A -85,B 0,C 180,E1 -3814.564,E2 -3814.564} C_VEL
LIN {X 0,Y 545.058,Z 381.216,A -85,B 0,C 180,E1 -3817.02,E2 -3817.02} C_VEL
LIN {X 0,Y 544.352,Z 381.304,A -85,B 0,C 180,E1 -3817.636,E2 -3817.636} C_VEL
LIN {X 0,Y 541.489,Z 381.659,A -85,B 0,C 180,E1 -3818.637,E2 -3818.637} C_VEL
LIN {X 0,Y 539.102,Z 381.958,A -85,B 0,C 180,E1 -3819.443,E2 -3819.443} C_VEL
LIN {X 0,Y 538.092,Z 382.08,A -85,B 0,C 180,E1 -3820.065,E2 -3820.065} C_VEL
LIN {X 0,Y 538.017,Z 382.089,A -85,B 0,C 180,E1 -3820.276,E2 -3820.276} C_VEL
LIN {X 0,Y 538.029,Z 382.094,A -85,B 0,C 180,E1 -3822.99,E2 -3822.99} C_VEL
LIN {X 0,Y 538.026,Z 382.088,A -85,B 0,C 180,E1 -3825.926,E2 -3825.926} C_VEL
LIN {X 0,Y 538.075,Z 382.087,A -85,B 0,C 180,E1 -3829.25,E2 -3829.25} C_VEL
LIN {X 0,Y 537.992,Z 382.092,A -85,B 0,C 180,E1 -3832.124,E2 -3832.124} C_VEL
LIN {X 0,Y 538.019,Z 382.095,A -85,B 0,C 180,E1 -3834.919,E2 -3834.919} C_VEL
LIN {X 0,Y 538.03,Z 382.089,A -85,B 0,C 180,E1 -3837.619,E2 -3837.619} C_VEL
LIN {X 0,Y 538.018,Z 382.089,A -85,B 0,C 180,E1 -3840.24,E2 -3840.24} C_VEL
LIN {X 0,Y 538.063,Z 382.089,A -85,B 0,C 180,E1 -3842.797,E2 -3842.797} C_VEL
LIN {X 0,Y 538.049,Z 382.089,A -85,B 0,C 180,E1 -3845.294,E2 -3845.294} C_VEL
LIN {X 0,Y 538.024,Z 382.091,A -85,B 0,C 180,E1 -3848.547,E2 -3848.547} C_VEL
LIN {X 0,Y 538.035,Z 382.093,A -85,B 0,C 180,E1 -3850.941,E2 -3850.941} C_VEL
LIN {X 0,Y 538.023,Z 382.092,A -85,B 0,C 180,E1 -3853.3,E2 -3853.3} C_VEL
LIN {X 0,Y 537.977,Z 382.098,A -85,B 0,C 180,E1 -3855.629,E2 -3855.629} C_VEL
LIN {X 0,Y 537.695,Z 382.136,A -85,B 0,C 180,E1 -3858.694,E2 -3858.694} C_VEL
LIN {X 0,Y 537.611,Z 382.286,A -85,B 0,C 180,E1 -3859.777,E2 -3859.777} C_VEL
LIN {X 0,Y 539.177,Z 391.671,A -85,B 0,C 180,E1 -3860.056,E2 -3860.056} C_VEL
LIN {X 0,Y 539.048,Z 403.76,A -85,B 0,C 180,E1 -3860.479,E2 -3860.479} C_VEL
LIN {X 0,Y 538.85,Z 414.667,A -85,B 0,C 180,E1 -3860.996,E2 -3860.996} C_VEL
LIN {X 0,Y 538.594,Z 425.557,A -85,B 0,C 180,E1 -3861.654,E2 -3861.654} C_VEL
LIN {X 0,Y 538.293,Z 436.71,A -85,B 0,C 180,E1 -3862.499,E2 -3862.499} C_VEL
LIN {X 0,Y 538.072,Z 446.67,A -85,B 0,C 180,E1 -3863.438,E2 -3863.438} C_VEL
LIN {X 0,Y 537.982,Z 456.221,A -85,B 0,C 180,E1 -3864.566,E2 -3864.566} C_VEL
LIN {X 0,Y 537.839,Z 463.93,A -85,B 0,C 180,E1 -3865.692,E2 -3865.692} C_VEL
LIN {X 0,Y 537.703,Z 469.162,A -85,B 0,C 180,E1 -3866.629,E2 -3866.629} C_VEL
LIN {X 0,Y 537.54,Z 474.286,A -85,B 0,C 180,E1 -3867.753,E2 -3867.753} C_VEL
LIN {X 0,Y 537.559,Z 478.256,A -85,B 0,C 180,E1 -3868.877,E2 -3868.877} C_VEL
LIN {X 0,Y 537.448,Z 481.196,A -85,B 0,C 180,E1 -3870.001,E2 -3870.001} C_VEL
LIN {X 0,Y 537.443,Z 482.628,A -85,B 0,C 180,E1 -3870.75,E2 -3870.75} C_VEL
LIN {X 0,Y 537.489,Z 484.255,A -85,B 0,C 180,E1 -3872.249,E2 -3872.249} C_VEL
LIN {X 0,Y 537.545,Z 484.496,A -85,B 0,C 180,E1 -3872.999,E2 -3872.999} C_VEL
LIN {X 0,Y 537.562,Z 484.313,A -85,B 0,C 180,E1 -3873.749,E2 -3873.749} C_VEL
LIN {X 0,Y 537.533,Z 482.758,A -85,B 0,C 180,E1 -3875.252,E2 -3875.252} C_VEL
LIN {X 0,Y 537.549,Z 480.321,A -85,B 0,C 180,E1 -3876.463,E2 -3876.463} C_VEL
LIN {X 0,Y 537.555,Z 477.283,A -85,B 0,C 180,E1 -3877.513,E2 -3877.513} C_VEL
LIN {X 0,Y 537.638,Z 472.979,A -85,B 0,C 180,E1 -3878.647,E2 -3878.647} C_VEL
LIN {X 0,Y 537.713,Z 467.474,A -85,B 0,C 180,E1 -3879.783,E2 -3879.783} C_VEL
LIN {X 0,Y 537.822,Z 460.564,A -85,B 0,C 180,E1 -3880.923,E2 -3880.923} C_VEL
LIN {X 0,Y 538.001,Z 451.892,A -85,B 0,C 180,E1 -3882.065,E2 -3882.065} C_VEL
LIN {X 0,Y 538.173,Z 442.025,A -85,B 0,C 180,E1 -3883.115,E2 -3883.115} C_VEL
LIN {X 0,Y 538.424,Z 431.957,A -85,B 0,C 180,E1 -3883.975,E2 -3883.975} C_VEL
LIN {X 0,Y 538.677,Z 421.147,A -85,B 0,C 180,E1 -3884.72,E2 -3884.72} C_VEL
LIN {X 0,Y 538.91,Z 409.176,A -85,B 0,C 180,E1 -3885.372,E2 -3885.372} C_VEL
LIN {X 0,Y 539.107,Z 396.311,A -85,B 0,C 180,E1 -3885.889,E2 -3885.889} C_VEL
LIN {X 0,Y 538.981,Z 390.044,A -85,B 0,C 180,E1 -3886.087,E2 -3886.087} C_VEL
LIN {X 0,Y 537.535,Z 382.155,A -85,B 0,C 180,E1 -3886.327,E2 -3886.327} C_VEL
LIN {X 0,Y 537.79,Z 382.122,A -85,B 0,C 180,E1 -3889.07,E2 -3889.07} C_VEL
LIN {X 0,Y 538.021,Z 382.088,A -85,B 0,C 180,E1 -3891.958,E2 -3891.958} C_VEL
LIN {X 0,Y 538.054,Z 382.087,A -85,B 0,C 180,E1 -3894.708,E2 -3894.708} C_VEL
LIN {X 0,Y 538.055,Z 382.087,A -85,B 0,C 180,E1 -3897.35,E2 -3897.35} C_VEL
LIN {X 0,Y 538.023,Z 382.088,A -85,B 0,C 180,E1 -3899.761,E2 -3899.761} C_VEL
LIN {X 0,Y 538.022,Z 382.091,A -85,B 0,C 180,E1 -3902.383,E2 -3902.383} C_VEL
LIN {X 0,Y 538.004,Z 382.094,A -85,B 0,C 180,E1 -3905.085,E2 -3905.085} C_VEL
LIN {X 0,Y 537.998,Z 382.089,A -85,B 0,C 180,E1 -3907.878,E2 -3907.878} C_VEL
LIN {X 0,Y 538.054,Z 382.088,A -85,B 0,C 180,E1 -3910.776,E2 -3910.776} C_VEL
LIN {X 0,Y 538.027,Z 382.09,A -85,B 0,C 180,E1 -3914.074,E2 -3914.074} C_VEL
LIN {X 0,Y 538.039,Z 382.086,A -85,B 0,C 180,E1 -3917.012,E2 -3917.012} C_VEL
LIN {X 0,Y 538.057,Z 382.081,A -85,B 0,C 180,E1 -3919.252,E2 -3919.252} C_VEL
LIN {X 0,Y 537.999,Z 382.09,A -85,B 0,C 180,E1 -3922.122,E2 -3922.122} C_VEL
LIN {X 0,Y 538.019,Z 382.088,A -85,B 0,C 180,E1 -3924.917,E2 -3924.917} C_VEL
LIN {X 0,Y 538.023,Z 382.09,A -85,B 0,C 180,E1 -3927.617,E2 -3927.617} C_VEL
LIN {X 0,Y 538.021,Z 382.081,A -85,B 0,C 180,E1 -3930.239,E2 -3930.239} C_VEL
LIN {X 0,Y 538.067,Z 382.078,A -85,B 0,C 180,E1 -3932.796,E2 -3932.796} C_VEL
LIN {X 0,Y 538.031,Z 382.089,A -85,B 0,C 180,E1 -3935.291,E2 -3935.291} C_VEL
LIN {X 0,Y 538.019,Z 382.091,A -85,B 0,C 180,E1 -3938.042,E2 -3938.042} C_VEL
LIN {X 0,Y 538.036,Z 382.087,A -85,B 0,C 180,E1 -3940.94,E2 -3940.94} C_VEL
LIN {X 0,Y 538.024,Z 382.095,A -85,B 0,C 180,E1 -3943.299,E2 -3943.299} C_VEL
LIN {X 0,Y 538.12,Z 382.202,A -85,B 0,C 180,E1 -3945.68,E2 -3945.68} C_VEL
LIN {X 0,Y 539.598,Z 387.909,A -85,B 0,C 180,E1 -3945.961,E2 -3945.961} C_VEL
LIN {X 0,Y 539.431,Z 398.159,A -85,B 0,C 180,E1 -3946.437,E2 -3946.437} C_VEL
LIN {X 0,Y 539.162,Z 408.283,A -85,B 0,C 180,E1 -3947.005,E2 -3947.005} C_VEL
LIN {X 0,Y 538.877,Z 418.161,A -85,B 0,C 180,E1 -3947.669,E2 -3947.669} C_VEL
LIN {X 0,Y 538.684,Z 426.917,A -85,B 0,C 180,E1 -3948.36,E2 -3948.36} C_VEL
LIN {X 0,Y 538.502,Z 434.941,A -85,B 0,C 180,E1 -3949.091,E2 -3949.091} C_VEL
LIN {X 0,Y 538.249,Z 442.206,A -85,B 0,C 180,E1 -3949.847,E2 -3949.847} C_VEL
LIN {X 0,Y 538.061,Z 450.023,A -85,B 0,C 180,E1 -3950.793,E2 -3950.793} C_VEL
LIN {X 0,Y 537.879,Z 457.932,A -85,B 0,C 180,E1 -3951.925,E2 -3951.925} C_VEL
LIN {X 0,Y 537.751,Z 463.529,A -85,B 0,C 180,E1 -3952.868,E2 -3952.868} C_VEL
LIN {X 0,Y 537.707,Z 469.19,A -85,B 0,C 180,E1 -3953.998,E2 -3953.998} C_VEL
LIN {X 0,Y 537.57,Z 473.835,A -85,B 0,C 180,E1 -3955.125,E2 -3955.125} C_VEL
LIN {X 0,Y 537.601,Z 477.562,A -85,B 0,C 180,E1 -3956.252,E2 -3956.252} C_VEL
LIN {X 0,Y 537.593,Z 479.636,A -85,B 0,C 180,E1 -3957.002,E2 -3957.002} C_VEL
LIN {X 0,Y 537.449,Z 482.529,A -85,B 0,C 180,E1 -3958.501,E2 -3958.501} C_VEL
LIN {X 0,Y 537.438,Z 483.55,A -85,B 0,C 180,E1 -3959.251,E2 -3959.251} C_VEL
LIN {X 0,Y 537.437,Z 484.429,A -85,B 0,C 180,E1 -3960.749,E2 -3960.749} C_VEL
LIN {X 0,Y 537.45,Z 484.425,A -85,B 0,C 180,E1 -3961.498,E2 -3961.498} C_VEL
LIN {X 0,Y 537.545,Z 483.364,A -85,B 0,C 180,E1 -3962.998,E2 -3962.998} C_VEL
LIN {X 0,Y 537.502,Z 480.904,A -85,B 0,C 180,E1 -3964.499,E2 -3964.499} C_VEL
LIN {X 0,Y 537.602,Z 478.172,A -85,B 0,C 180,E1 -3965.627,E2 -3965.627} C_VEL
LIN {X 0,Y 537.618,Z 474.597,A -85,B 0,C 180,E1 -3966.756,E2 -3966.756} C_VEL
LIN {X 0,Y 537.668,Z 470.106,A -85,B 0,C 180,E1 -3967.888,E2 -3967.888} C_VEL
LIN {X 0,Y 537.775,Z 464.6,A -85,B 0,C 180,E1 -3969.022,E2 -3969.022} C_VEL
LIN {X 0,Y 537.862,Z 459.167,A -85,B 0,C 180,E1 -3969.97,E2 -3969.97} C_VEL
LIN {X 0,Y 538.021,Z 452.827,A -85,B 0,C 180,E1 -3970.918,E2 -3970.918} C_VEL
LIN {X 0,Y 538.183,Z 445.113,A -85,B 0,C 180,E1 -3971.905,E2 -3971.905} C_VEL
LIN {X 0,Y 538.395,Z 436.725,A -85,B 0,C 180,E1 -3972.821,E2 -3972.821} C_VEL
LIN {X 0,Y 538.611,Z 428.622,A -85,B 0,C 180,E1 -3973.584,E2 -3973.584} C_VEL
LIN {X 0,Y 538.872,Z 419.16,A -85,B 0,C 180,E1 -3974.347,E2 -3974.347} C_VEL
LIN {X 0,Y 539.126,Z 409.385,A -85,B 0,C 180,E1 -3975.016,E2 -3975.016} C_VEL
LIN {X 0,Y 539.398,Z 399.114,A -85,B 0,C 180,E1 -3975.604,E2 -3975.604} C_VEL
LIN {X 0,Y 539.573,Z 389.34,A -85,B 0,C 180,E1 -3976.068,E2 -3976.068} C_VEL
LIN {X 0,Y 539.097,Z 386.026,A -85,B 0,C 180,E1 -3976.229,E2 -3976.229} C_VEL
LIN {X 0,Y 538.063,Z 382.091,A -85,B 0,C 180,E1 -3976.431,E2 -3976.431} C_VEL
LIN {X 0,Y 538.043,Z 382.093,A -85,B 0,C 180,E1 -3979.06,E2 -3979.06} C_VEL
LIN {X 0,Y 538.018,Z 382.095,A -85,B 0,C 180,E1 -3981.958,E2 -3981.958} C_VEL
LIN {X 0,Y 538.052,Z 382.09,A -85,B 0,C 180,E1 -3984.707,E2 -3984.707} C_VEL
LIN {X 0,Y 538.062,Z 382.088,A -85,B 0,C 180,E1 -3987.352,E2 -3987.352} C_VEL
LIN {X 0,Y 538.019,Z 382.093,A -85,B 0,C 180,E1 -3989.761,E2 -3989.761} C_VEL
LIN {X 0,Y 538.029,Z 382.092,A -85,B 0,C 180,E1 -3992.382,E2 -3992.382} C_VEL
LIN {X 0,Y 538.001,Z 382.097,A -85,B 0,C 180,E1 -3995.084,E2 -3995.084} C_VEL
LIN {X 0,Y 537.995,Z 382.098,A -85,B 0,C 180,E1 -3997.877,E2 -3997.877} C_VEL
LIN {X 0,Y 538.052,Z 382.09,A -85,B 0,C 180,E1 -4000.775,E2 -4000.775} C_VEL
LIN {X 0,Y 538.033,Z 382.095,A -85,B 0,C 180,E1 -4004.074,E2 -4004.074} C_VEL
LIN {X 0,Y 538.022,Z 382.095,A -85,B 0,C 180,E1 -4007.214,E2 -4007.214} C_VEL
LIN {X 0,Y 538.03,Z 382.095,A -85,B 0,C 180,E1 -4010.203,E2 -4010.203} C_VEL
LIN {X 0,Y 538.087,Z 382.282,A -85,B 0,C 180,E1 -4010.693,E2 -4010.693} C_VEL
LIN {X 0,Y 538.791,Z 387.139,A -85,B 0,C 180,E1 -4011.862,E2 -4011.862} C_VEL
LIN {X 0,Y 538.496,Z 398.243,A -85,B 0,C 180,E1 -4014.264,E2 -4014.264} C_VEL
LIN {X 0,Y 538.479,Z 414.949,A -85,B 0,C 180,E1 -4017.648,E2 -4017.648} C_VEL
LIN {X 0,Y 538.648,Z 428.528,A -85,B 0,C 180,E1 -4020.277,E2 -4020.277} C_VEL
LIN {X 0,Y 538.654,Z 444.307,A -85,B 0,C 180,E1 -4023.247,E2 -4023.247} C_VEL
LIN {X 0,Y 538.65,Z 458.939,A -85,B 0,C 180,E1 -4025.968,E2 -4025.968} C_VEL
LIN {X 0,Y 538.535,Z 475.184,A -85,B 0,C 180,E1 -4028.968,E2 -4028.968} C_VEL
LIN {X 0,Y 538.426,Z 485.645,A -85,B 0,C 180,E1 -4030.954,E2 -4030.954} C_VEL
LIN {X 0,Y 538.189,Z 499.039,A -85,B 0,C 180,E1 -4033.694,E2 -4033.694} C_VEL
LIN {X 0,Y 538.169,Z 499.756,A -85,B 0,C 180,E1 -4033.839,E2 -4033.839} C_VEL
LIN {X 0,Y 540.105,Z 510.134,A -85,B 0,C 180,E1 -4034.074,E2 -4034.074} C_VEL
LIN {X 0,Y 539.861,Z 524.316,A -85,B 0,C 180,E1 -4034.423,E2 -4034.423} C_VEL
LIN {X 0,Y 539.619,Z 538.81,A -85,B 0,C 180,E1 -4034.949,E2 -4034.949} C_VEL
LIN {X 0,Y 539.364,Z 551.627,A -85,B 0,C 180,E1 -4035.569,E2 -4035.569} C_VEL
LIN {X 0,Y 538.989,Z 564.092,A -85,B 0,C 180,E1 -4036.329,E2 -4036.329} C_VEL
LIN {X 0,Y 538.704,Z 576.637,A -85,B 0,C 180,E1 -4037.281,E2 -4037.281} C_VEL
LIN {X 0,Y 538.435,Z 586.813,A -85,B 0,C 180,E1 -4038.223,E2 -4038.223} C_VEL
LIN {X 0,Y 538.205,Z 596.327,A -85,B 0,C 180,E1 -4039.275,E2 -4039.275} C_VEL
LIN {X 0,Y 537.969,Z 604.905,A -85,B 0,C 180,E1 -4040.411,E2 -4040.411} C_VEL
LIN {X 0,Y 537.805,Z 613.115,A -85,B 0,C 180,E1 -4041.735,E2 -4041.735} C_VEL
LIN {X 0,Y 537.661,Z 618.859,A -85,B 0,C 180,E1 -4042.866,E2 -4042.866} C_VEL
LIN {X 0,Y 537.656,Z 624.958,A -85,B 0,C 180,E1 -4044.373,E2 -4044.373} C_VEL
LIN {X 0,Y 537.55,Z 628.444,A -85,B 0,C 180,E1 -4045.5,E2 -4045.5} C_VEL
LIN {X 0,Y 537.547,Z 631.833,A -85,B 0,C 180,E1 -4047.001,E2 -4047.001} C_VEL
LIN {X 0,Y 537.447,Z 633.834,A -85,B 0,C 180,E1 -4048.501,E2 -4048.501} C_VEL
LIN {X 0,Y 537.44,Z 634.5,A -85,B 0,C 180,E1 -4049.999,E2 -4049.999} C_VEL
LIN {X 0,Y 537.447,Z 633.835,A -85,B 0,C 180,E1 -4051.498,E2 -4051.498} C_VEL
LIN {X 0,Y 537.547,Z 631.834,A -85,B 0,C 180,E1 -4052.997,E2 -4052.997} C_VEL
LIN {X 0,Y 537.55,Z 628.446,A -85,B 0,C 180,E1 -4054.498,E2 -4054.498} C_VEL
LIN {X 0,Y 537.649,Z 623.572,A -85,B 0,C 180,E1 -4056.002,E2 -4056.002} C_VEL
LIN {X 0,Y 537.703,Z 617.059,A -85,B 0,C 180,E1 -4057.509,E2 -4057.509} C_VEL
LIN {X 0,Y 537.858,Z 609.807,A -85,B 0,C 180,E1 -4058.831,E2 -4058.831} C_VEL
LIN {X 0,Y 538.062,Z 600.829,A -85,B 0,C 180,E1 -4060.155,E2 -4060.155} C_VEL
LIN {X 0,Y 538.341,Z 591.401,A -85,B 0,C 180,E1 -4061.292,E2 -4061.292} C_VEL
LIN {X 0,Y 538.56,Z 580.965,A -85,B 0,C 180,E1 -4062.338,E2 -4062.338} C_VEL
LIN {X 0,Y 538.869,Z 569.442,A -85,B 0,C 180,E1 -4063.288,E2 -4063.288} C_VEL
LIN {X 0,Y 539.23,Z 556.653,A -85,B 0,C 180,E1 -4064.144,E2 -4064.144} C_VEL
LIN {X 0,Y 539.518,Z 544.173,A -85,B 0,C 180,E1 -4064.811,E2 -4064.811} C_VEL
LIN {X 0,Y 539.799,Z 531.044,A -85,B 0,C 180,E1 -4065.354,E2 -4065.354} C_VEL
LIN {X 0,Y 539.98,Z 516.864,A -85,B 0,C 180,E1 -4065.781,E2 -4065.781} C_VEL
LIN {X 0,Y 539.955,Z 509.351,A -85,B 0,C 180,E1 -4065.947,E2 -4065.947} C_VEL
LIN {X 0,Y 538.165,Z 499.764,A -85,B 0,C 180,E1 -4066.159,E2 -4066.159} C_VEL
LIN {X 0,Y 538.402,Z 487.572,A -85,B 0,C 180,E1 -4068.65,E2 -4068.65} C_VEL
LIN {X 0,Y 538.576,Z 474.51,A -85,B 0,C 180,E1 -4071.229,E2 -4071.229} C_VEL
LIN {X 0,Y 538.72,Z 460.217,A -85,B 0,C 180,E1 -4074.048,E2 -4074.048} C_VEL
LIN {X 0,Y 538.944,Z 447.137,A -85,B 0,C 180,E1 -4076.735,E2 -4076.735} C_VEL
LIN {X 0,Y 539.189,Z 431.986,A -85,B 0,C 180,E1 -4079.904,E2 -4079.904} C_VEL
LIN {X 0,Y 539.411,Z 416.907,A -85,B 0,C 180,E1 -4083.175,E2 -4083.175} C_VEL
LIN {X 0,Y 539.842,Z 400.955,A -85,B 0,C 180,E1 -4086.787,E2 -4086.787} C_VEL
LIN {X 0,Y 540.062,Z 392.947,A -85,B 0,C 180,E1 -4088.666,E2 -4088.666} C_VEL
LIN {X 0,Y 538.986,Z 386.575,A -85,B 0,C 180,E1 -4090.289,E2 -4090.289} C_VEL
LIN {X 0,Y 538.058,Z 382.089,A -85,B 0,C 180,E1 -4091.518,E2 -4091.518} C_VEL
LIN {X 0,Y 538.022,Z 382.095,A -85,B 0,C 180,E1 -4094.074,E2 -4094.074} C_VEL
LIN {X 0,Y 538.018,Z 382.09,A -85,B 0,C 180,E1 -4097.214,E2 -4097.214} C_VEL
LIN {X 0,Y 538.047,Z 382.087,A -85,B 0,C 180,E1 -4100.205,E2 -4100.205} C_VEL
LIN {X 0,Y 538.025,Z 382.088,A -85,B 0,C 180,E1 -4103.067,E2 -4103.067} C_VEL
LIN {X 0,Y 538.024,Z 382.093,A -85,B 0,C 180,E1 -4105.827,E2 -4105.827} C_VEL
LIN {X 0,Y 538.015,Z 382.089,A -85,B 0,C 180,E1 -4108.499,E2 -4108.499} C_VEL
LIN {X 0,Y 538.049,Z 382.086,A -85,B 0,C 180,E1 -4111.099,E2 -4111.099} C_VEL
LIN {X 0,Y 538.041,Z 382.092,A -85,B 0,C 180,E1 -4113.633,E2 -4113.633} C_VEL
LIN {X 0,Y 538.012,Z 382.092,A -85,B 0,C 180,E1 -4116.118,E2 -4116.118} C_VEL
LIN {X 0,Y 538.033,Z 382.092,A -85,B 0,C 180,E1 -4119.348,E2 -4119.348} C_VEL
LIN {X 0,Y 538.062,Z 382.083,A -85,B 0,C 180,E1 -4122.517,E2 -4122.517} C_VEL
LIN {X 0,Y 538.053,Z 382.09,A -85,B 0,C 180,E1 -4125.631,E2 -4125.631} C_VEL
LIN {X 0,Y 538.079,Z 382.081,A -85,B 0,C 180,E1 -4128.702,E2 -4128.702} C_VEL
LIN {X 0,Y 538.081,Z 382.086,A -85,B 0,C 180,E1 -4131.74,E2 -4131.74} C_VEL
LIN {X 0,Y 538.156,Z 382.072,A -85,B 0,C 180,E1 -4134.755,E2 -4134.755} C_VEL
LIN {X 0,Y 538.158,Z 382.076,A -85,B 0,C 180,E1 -4137.755,E2 -4137.755} C_VEL
LIN {X 0,Y 538.177,Z 382.069,A -85,B 0,C 180,E1 -4140.748,E2 -4140.748} C_VEL
LIN {X 0,Y 538.134,Z 382.077,A -85,B 0,C 180,E1 -4142.995,E2 -4142.995} C_VEL
LIN {X 0,Y 538.115,Z 382.078,A -85,B 0,C 180,E1 -4145.998,E2 -4145.998} C_VEL
LIN {X 0,Y 538.068,Z 382.086,A -85,B 0,C 180,E1 -4149.018,E2 -4149.018} C_VEL
LIN {X 0,Y 538.074,Z 382.082,A -85,B 0,C 180,E1 -4152.063,E2 -4152.063} C_VEL
LIN {X 0,Y 538.036,Z 382.092,A -85,B 0,C 180,E1 -4155.144,E2 -4155.144} C_VEL
LIN {X 0,Y 538.026,Z 382.087,A -85,B 0,C 180,E1 -4158.271,E2 -4158.271} C_VEL
LIN {X 0,Y 538.034,Z 382.087,A -85,B 0,C 180,E1 -4160.652,E2 -4160.652} C_VEL
LIN {X 0,Y 538.015,Z 382.09,A -85,B 0,C 180,E1 -4163.888,E2 -4163.888} C_VEL
LIN {X 0,Y 538.043,Z 382.085,A -85,B 0,C 180,E1 -4166.367,E2 -4166.367} C_VEL
LIN {X 0,Y 538.024,Z 382.092,A -85,B 0,C 180,E1 -4168.935,E2 -4168.935} C_VEL
LIN {X 0,Y 538.021,Z 382.089,A -85,B 0,C 180,E1 -4171.891,E2 -4171.891} C_VEL
LIN {X 0,Y 538.027,Z 382.089,A -85,B 0,C 180,E1 -4174.622,E2 -4174.622} C_VEL
LIN {X 0,Y 538.002,Z 382.097,A -85,B 0,C 180,E1 -4177.172,E2 -4177.172} C_VEL
LIN {X 0,Y 538.017,Z 382.089,A -85,B 0,C 180,E1 -4180.276,E2 -4180.276} C_VEL
LIN {X 0,Y 537.367,Z 382.175,A -85,B 0,C 180,E1 -4180.901,E2 -4180.901} C_VEL
LIN {X 0,Y 534.519,Z 382.532,A -85,B 0,C 180,E1 -4181.916,E2 -4181.916} C_VEL
LIN {X 0,Y 532.095,Z 382.835,A -85,B 0,C 180,E1 -4182.733,E2 -4182.733} C_VEL
LIN {X 0,Y 531.048,Z 382.962,A -85,B 0,C 180,E1 -4183.364,E2 -4183.364} C_VEL
LIN {X 0,Y 530.96,Z 382.971,A -85,B 0,C 180,E1 -4183.578,E2 -4183.578} C_VEL
LIN {X 0,Y 530.961,Z 382.969,A -85,B 0,C 180,E1 -4186.507,E2 -4186.507} C_VEL
LIN {X 0,Y 531.005,Z 382.965,A -85,B 0,C 180,E1 -4189.571,E2 -4189.571} C_VEL
LIN {X 0,Y 530.967,Z 382.969,A -85,B 0,C 180,E1 -4192.578,E2 -4192.578} C_VEL
LIN {X 0,Y 531,Z 382.968,A -85,B 0,C 180,E1 -4195.312,E2 -4195.312} C_VEL
LIN {X 0,Y 530.982,Z 382.965,A -85,B 0,C 180,E1 -4198.034,E2 -4198.034} C_VEL
LIN {X 0,Y 530.989,Z 382.971,A -85,B 0,C 180,E1 -4200.875,E2 -4200.875} C_VEL
LIN {X 0,Y 531.005,Z 382.967,A -85,B 0,C 180,E1 -4203.258,E2 -4203.258} C_VEL
LIN {X 0,Y 530.986,Z 382.964,A -85,B 0,C 180,E1 -4205.962,E2 -4205.962} C_VEL
LIN {X 0,Y 531,Z 382.968,A -85,B 0,C 180,E1 -4209.063,E2 -4209.063} C_VEL
LIN {X 0,Y 530.99,Z 382.966,A -85,B 0,C 180,E1 -4211.48,E2 -4211.48} C_VEL
LIN {X 0,Y 530.975,Z 382.966,A -85,B 0,C 180,E1 -4213.863,E2 -4213.863} C_VEL
LIN {X 0,Y 530.837,Z 382.991,A -85,B 0,C 180,E1 -4216.214,E2 -4216.214} C_VEL
LIN {X 0,Y 530.67,Z 383.01,A -85,B 0,C 180,E1 -4218.543,E2 -4218.543} C_VEL
LIN {X 0,Y 530.547,Z 383.024,A -85,B 0,C 180,E1 -4219.579,E2 -4219.579} C_VEL
LIN {X 0,Y 532.329,Z 392.361,A -85,B 0,C 180,E1 -4219.878,E2 -4219.878} C_VEL
LIN {X 0,Y 532.203,Z 404.531,A -85,B 0,C 180,E1 -4220.308,E2 -4220.308} C_VEL
LIN {X 0,Y 531.947,Z 416.348,A -85,B 0,C 180,E1 -4220.879,E2 -4220.879} C_VEL
LIN {X 0,Y 531.638,Z 428.341,A -85,B 0,C 180,E1 -4221.64,E2 -4221.64} C_VEL
LIN {X 0,Y 531.341,Z 439.163,A -85,B 0,C 180,E1 -4222.513,E2 -4222.513} C_VEL
LIN {X 0,Y 531.04,Z 449.38,A -85,B 0,C 180,E1 -4223.552,E2 -4223.552} C_VEL
LIN {X 0,Y 530.953,Z 456.89,A -85,B 0,C 180,E1 -4224.494,E2 -4224.494} C_VEL
LIN {X 0,Y 530.789,Z 464.37,A -85,B 0,C 180,E1 -4225.635,E2 -4225.635} C_VEL
LIN {X 0,Y 530.635,Z 469.447,A -85,B 0,C 180,E1 -4226.584,E2 -4226.584} C_VEL
LIN {X 0,Y 530.462,Z 474.452,A -85,B 0,C 180,E1 -4227.723,E2 -4227.723} C_VEL
LIN {X 0,Y 530.478,Z 478.383,A -85,B 0,C 180,E1 -4228.862,E2 -4228.862} C_VEL
LIN {X 0,Y 530.349,Z 481.29,A -85,B 0,C 180,E1 -4230.001,E2 -4230.001} C_VEL
LIN {X 0,Y 530.345,Z 482.687,A -85,B 0,C 180,E1 -4230.76,E2 -4230.76} C_VEL
LIN {X 0,Y 530.41,Z 484.28,A -85,B 0,C 180,E1 -4232.279,E2 -4232.279} C_VEL
LIN {X 0,Y 530.45,Z 484.5,A -85,B 0,C 180,E1 -4233.039,E2 -4233.039} C_VEL
LIN {X 0,Y 530.48,Z 484.288,A -85,B 0,C 180,E1 -4233.799,E2 -4233.799} C_VEL
LIN {X 0,Y 530.456,Z 482.698,A -85,B 0,C 180,E1 -4235.322,E2 -4235.322} C_VEL
LIN {X 0,Y 530.469,Z 480.44,A -85,B 0,C 180,E1 -4236.457,E2 -4236.457} C_VEL
LIN {X 0,Y 530.469,Z 477.151,A -85,B 0,C 180,E1 -4237.614,E2 -4237.614} C_VEL
LIN {X 0,Y 530.56,Z 472.806,A -85,B 0,C 180,E1 -4238.763,E2 -4238.763} C_VEL
LIN {X 0,Y 530.694,Z 466.342,A -85,B 0,C 180,E1 -4240.107,E2 -4240.107} C_VEL
LIN {X 0,Y 530.839,Z 459.267,A -85,B 0,C 180,E1 -4241.262,E2 -4241.262} C_VEL
LIN {X 0,Y 531.047,Z 450.423,A -85,B 0,C 180,E1 -4242.42,E2 -4242.42} C_VEL
LIN {X 0,Y 531.321,Z 440.176,A -85,B 0,C 180,E1 -4243.482,E2 -4243.482} C_VEL
LIN {X 0,Y 531.589,Z 429.724,A -85,B 0,C 180,E1 -4244.353,E2 -4244.353} C_VEL
LIN {X 0,Y 531.923,Z 417.779,A -85,B 0,C 180,E1 -4245.13,E2 -4245.13} C_VEL
LIN {X 0,Y 532.123,Z 406.268,A -85,B 0,C 180,E1 -4245.71,E2 -4245.71} C_VEL
LIN {X 0,Y 532.276,Z 393.771,A -85,B 0,C 180,E1 -4246.172,E2 -4246.172} C_VEL
LIN {X 0,Y 531.972,Z 389.97,A -85,B 0,C 180,E1 -4246.293,E2 -4246.293} C_VEL
LIN {X 0,Y 530.508,Z 383.03,A -85,B 0,C 180,E1 -4246.5,E2 -4246.5} C_VEL
LIN {X 0,Y 530.769,Z 382.996,A -85,B 0,C 180,E1 -4249.332,E2 -4249.332} C_VEL
LIN {X 0,Y 530.983,Z 382.965,A -85,B 0,C 180,E1 -4252.102,E2 -4252.102} C_VEL
LIN {X 0,Y 531.011,Z 382.967,A -85,B 0,C 180,E1 -4255.058,E2 -4255.058} C_VEL
LIN {X 0,Y 531.019,Z 382.961,A -85,B 0,C 180,E1 -4257.596,E2 -4257.596} C_VEL
LIN {X 0,Y 530.98,Z 382.971,A -85,B 0,C 180,E1 -4260.645,E2 -4260.645} C_VEL
LIN {X 0,Y 530.962,Z 382.968,A -85,B 0,C 180,E1 -4263.775,E2 -4263.775} C_VEL
LIN {X 0,Y 530.961,Z 382.975,A -85,B 0,C 180,E1 -4266.559,E2 -4266.559} C_VEL
LIN {X 0,Y 530.991,Z 382.962,A -85,B 0,C 180,E1 -4269.443,E2 -4269.443} C_VEL
LIN {X 0,Y 530.983,Z 382.971,A -85,B 0,C 180,E1 -4272.457,E2 -4272.457} C_VEL
LIN {X 0,Y 530.994,Z 382.962,A -85,B 0,C 180,E1 -4275.621,E2 -4275.621} C_VEL
LIN {X 0,Y 531.006,Z 382.964,A -85,B 0,C 180,E1 -4278.565,E2 -4278.565} C_VEL
LIN {X 0,Y 530.964,Z 382.959,A -85,B 0,C 180,E1 -4281.529,E2 -4281.529} C_VEL
LIN {X 0,Y 530.983,Z 382.968,A -85,B 0,C 180,E1 -4284.382,E2 -4284.382} C_VEL
LIN {X 0,Y 530.971,Z 382.964,A -85,B 0,C 180,E1 -4287.133,E2 -4287.133} C_VEL
LIN {X 0,Y 530.974,Z 382.962,A -85,B 0,C 180,E1 -4289.803,E2 -4289.803} C_VEL
LIN {X 0,Y 531.019,Z 382.957,A -85,B 0,C 180,E1 -4292.467,E2 -4292.467} C_VEL
LIN {X 0,Y 530.998,Z 382.962,A -85,B 0,C 180,E1 -4294.942,E2 -4294.942} C_VEL
LIN {X 0,Y 530.975,Z 382.966,A -85,B 0,C 180,E1 -4298.247,E2 -4298.247} C_VEL
LIN {X 0,Y 530.996,Z 382.963,A -85,B 0,C 180,E1 -4300.677,E2 -4300.677} C_VEL
LIN {X 0,Y 530.979,Z 382.969,A -85,B 0,C 180,E1 -4303.07,E2 -4303.07} C_VEL
LIN {X 0,Y 531.053,Z 382.964,A -85,B 0,C 180,E1 -4305.461,E2 -4305.461} C_VEL
LIN {X 0,Y 532.673,Z 388.804,A -85,B 0,C 180,E1 -4305.774,E2 -4305.774} C_VEL
LIN {X 0,Y 532.586,Z 398.953,A -85,B 0,C 180,E1 -4306.259,E2 -4306.259} C_VEL
LIN {X 0,Y 532.293,Z 408.975,A -85,B 0,C 180,E1 -4306.835,E2 -4306.835} C_VEL
LIN {X 0,Y 531.962,Z 418.736,A -85,B 0,C 180,E1 -4307.506,E2 -4307.506} C_VEL
LIN {X 0,Y 531.767,Z 426.869,A -85,B 0,C 180,E1 -4308.162,E2 -4308.162} C_VEL
LIN {X 0,Y 531.532,Z 435.256,A -85,B 0,C 180,E1 -4308.947,E2 -4308.947} C_VEL
LIN {X 0,Y 531.253,Z 442.39,A -85,B 0,C 180,E1 -4309.712,E2 -4309.712} C_VEL
LIN {X 0,Y 531.004,Z 451.516,A -85,B 0,C 180,E1 -4310.861,E2 -4310.861} C_VEL
LIN {X 0,Y 530.836,Z 458.013,A -85,B 0,C 180,E1 -4311.817,E2 -4311.817} C_VEL
LIN {X 0,Y 530.679,Z 463.599,A -85,B 0,C 180,E1 -4312.772,E2 -4312.772} C_VEL
LIN {X 0,Y 530.626,Z 469.245,A -85,B 0,C 180,E1 -4313.917,E2 -4313.917} C_VEL
LIN {X 0,Y 530.484,Z 473.879,A -85,B 0,C 180,E1 -4315.06,E2 -4315.06} C_VEL
LIN {X 0,Y 530.527,Z 477.596,A -85,B 0,C 180,E1 -4316.202,E2 -4316.202} C_VEL
LIN {X 0,Y 530.496,Z 479.667,A -85,B 0,C 180,E1 -4316.962,E2 -4316.962} C_VEL
LIN {X 0,Y 530.358,Z 482.542,A -85,B 0,C 180,E1 -4318.481,E2 -4318.481} C_VEL
LIN {X 0,Y 530.34,Z 483.567,A -85,B 0,C 180,E1 -4319.241,E2 -4319.241} C_VEL
LIN {X 0,Y 530.339,Z 484.422,A -85,B 0,C 180,E1 -4320.759,E2 -4320.759} C_VEL
LIN {X 0,Y 530.359,Z 484.421,A -85,B 0,C 180,E1 -4321.518,E2 -4321.518} C_VEL
LIN {X 0,Y 530.449,Z 483.339,A -85,B 0,C 180,E1 -4323.038,E2 -4323.038} C_VEL
LIN {X 0,Y 530.407,Z 480.868,A -85,B 0,C 180,E1 -4324.56,E2 -4324.56} C_VEL
LIN {X 0,Y 530.51,Z 478.126,A -85,B 0,C 180,E1 -4325.702,E2 -4325.702} C_VEL
LIN {X 0,Y 530.549,Z 474.539,A -85,B 0,C 180,E1 -4326.847,E2 -4326.847} C_VEL
LIN {X 0,Y 530.581,Z 470.036,A -85,B 0,C 180,E1 -4327.995,E2 -4327.995} C_VEL
LIN {X 0,Y 530.712,Z 464.52,A -85,B 0,C 180,E1 -4329.144,E2 -4329.144} C_VEL
LIN {X 0,Y 530.824,Z 459.07,A -85,B 0,C 180,E1 -4330.103,E2 -4330.103} C_VEL
LIN {X 0,Y 530.983,Z 452.714,A -85,B 0,C 180,E1 -4331.065,E2 -4331.065} C_VEL
LIN {X 0,Y 531.225,Z 443.757,A -85,B 0,C 180,E1 -4332.22,E2 -4332.22} C_VEL
LIN {X 0,Y 531.499,Z 434.982,A -85,B 0,C 180,E1 -4333.185,E2 -4333.185} C_VEL
LIN {X 0,Y 531.876,Z 423.334,A -85,B 0,C 180,E1 -4334.247,E2 -4334.247} C_VEL
LIN {X 0,Y 532.26,Z 411.354,A -85,B 0,C 180,E1 -4335.116,E2 -4335.116} C_VEL
LIN {X 0,Y 532.491,Z 402.448,A -85,B 0,C 180,E1 -4335.659,E2 -4335.659} C_VEL
LIN {X 0,Y 532.795,Z 390.928,A -85,B 0,C 180,E1 -4336.229,E2 -4336.229} C_VEL
LIN {X 0,Y 532.328,Z 387.632,A -85,B 0,C 180,E1 -4336.391,E2 -4336.391} C_VEL
LIN {X 0,Y 530.995,Z 382.971,A -85,B 0,C 180,E1 -4336.632,E2 -4336.632} C_VEL
LIN {X 0,Y 531,Z 382.97,A -85,B 0,C 180,E1 -4339.322,E2 -4339.322} C_VEL
LIN {X 0,Y 530.981,Z 382.971,A -85,B 0,C 180,E1 -4342.102,E2 -4342.102} C_VEL
LIN {X 0,Y 531.009,Z 382.969,A -85,B 0,C 180,E1 -4345.057,E2 -4345.057} C_VEL
LIN {X 0,Y 531.019,Z 382.967,A -85,B 0,C 180,E1 -4347.595,E2 -4347.595} C_VEL
LIN {X 0,Y 530.977,Z 382.971,A -85,B 0,C 180,E1 -4350.645,E2 -4350.645} C_VEL
LIN {X 0,Y 530.99,Z 382.969,A -85,B 0,C 180,E1 -4353.772,E2 -4353.772} C_VEL
LIN {X 0,Y 530.958,Z 382.975,A -85,B 0,C 180,E1 -4356.558,E2 -4356.558} C_VEL
LIN {X 0,Y 530.989,Z 382.97,A -85,B 0,C 180,E1 -4359.443,E2 -4359.443} C_VEL
LIN {X 0,Y 530.983,Z 382.971,A -85,B 0,C 180,E1 -4362.456,E2 -4362.456} C_VEL
LIN {X 0,Y 530.984,Z 382.972,A -85,B 0,C 180,E1 -4365.621,E2 -4365.621} C_VEL
LIN {X 0,Y 531,Z 382.97,A -85,B 0,C 180,E1 -4368.564,E2 -4368.564} C_VEL
LIN {X 0,Y 531.043,Z 383.092,A -85,B 0,C 180,E1 -4370.459,E2 -4370.459} C_VEL
LIN {X 0,Y 531.871,Z 388.664,A -85,B 0,C 180,E1 -4371.842,E2 -4371.842} C_VEL
LIN {X 0,Y 531.473,Z 400.357,A -85,B 0,C 180,E1 -4374.419,E2 -4374.419} C_VEL
LIN {X 0,Y 531.476,Z 416.818,A -85,B 0,C 180,E1 -4377.812,E2 -4377.812} C_VEL
LIN {X 0,Y 531.596,Z 431.815,A -85,B 0,C 180,E1 -4380.757,E2 -4380.757} C_VEL
LIN {X 0,Y 531.589,Z 447.2,A -85,B 0,C 180,E1 -4383.694,E2 -4383.694} C_VEL
LIN {X 0,Y 531.553,Z 461.73,A -85,B 0,C 180,E1 -4386.429,E2 -4386.429} C_VEL
LIN {X 0,Y 531.405,Z 476.977,A -85,B 0,C 180,E1 -4389.281,E2 -4389.281} C_VEL
LIN {X 0,Y 531.297,Z 489.967,A -85,B 0,C 180,E1 -4391.709,E2 -4391.709} C_VEL
LIN {X 0,Y 531.179,Z 499.881,A -85,B 0,C 180,E1 -4393.633,E2 -4393.633} C_VEL
LIN {X 0,Y 533.262,Z 510.987,A -85,B 0,C 180,E1 -4393.883,E2 -4393.883} C_VEL
LIN {X 0,Y 533.025,Z 525.049,A -85,B 0,C 180,E1 -4394.242,E2 -4394.242} C_VEL
LIN {X 0,Y 532.775,Z 538.808,A -85,B 0,C 180,E1 -4394.751,E2 -4394.751} C_VEL
LIN {X 0,Y 532.479,Z 551.625,A -85,B 0,C 180,E1 -4395.378,E2 -4395.378} C_VEL
LIN {X 0,Y 532.066,Z 564.09,A -85,B 0,C 180,E1 -4396.148,E2 -4396.148} C_VEL
LIN {X 0,Y 531.721,Z 576.639,A -85,B 0,C 180,E1 -4397.111,E2 -4397.111} C_VEL
LIN {X 0,Y 531.419,Z 587.532,A -85,B 0,C 180,E1 -4398.139,E2 -4398.139} C_VEL
LIN {X 0,Y 531.13,Z 597.847,A -85,B 0,C 180,E1 -4399.324,E2 -4399.324} C_VEL
LIN {X 0,Y 530.928,Z 606.17,A -85,B 0,C 180,E1 -4400.475,E2 -4400.475} C_VEL
LIN {X 0,Y 530.71,Z 614.124,A -85,B 0,C 180,E1 -4401.815,E2 -4401.815} C_VEL
